RoboDK station: kr30 cnc 101019.rdk

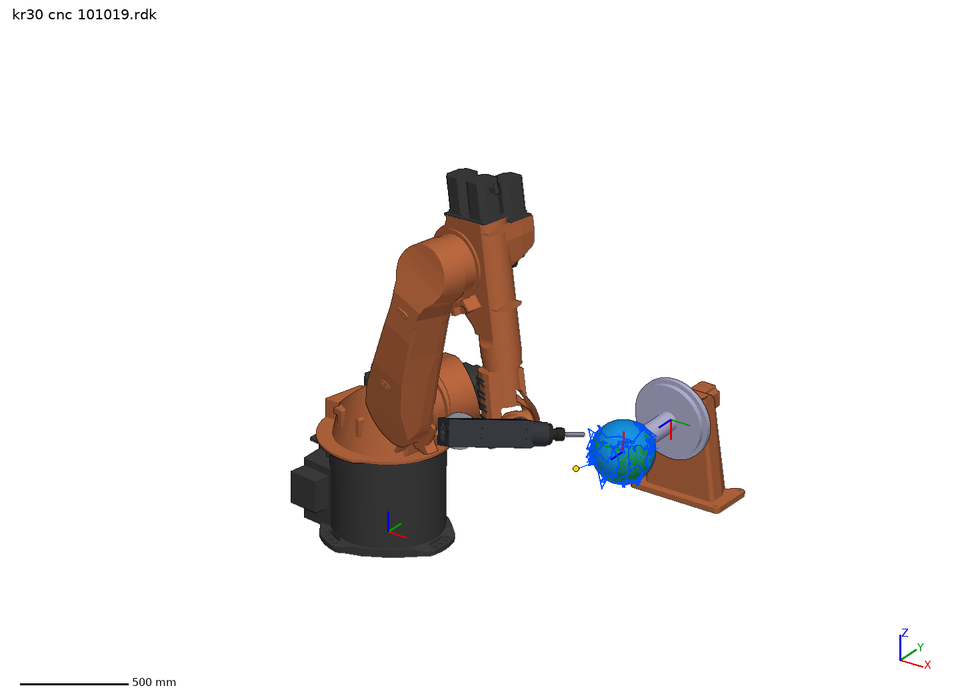
[picture v0: the station drawn from its stored meshes, robots at their saved joint values, targets as dots, program paths as lines]
Station kr30 cnc 101019. Poses are relative to the parent item; angles as X-Y-Z fixed-axis rotations.
  - frame KUKA KR 30 HA Base at (0, 0, 0) mm
    - robot KUKA KR 30 HA: 6 axes, payload 30 kg, reach 2033 mm, repeatability 0.05 mm, weight 665 kg
        modified DH rows (alpha deg, a mm, theta deg, d mm): 0, 0, 0, 815; -90, 350, 0, 0; 0, 850, -90, 0; -90, 145, 0, 820; 90, 0, 0, 0; -90, 0, 180, 170
        joint limits [-185, -135, -120, -350, -119, -350] to [185, 35, 158, 350, 119, 350]; home [0, -90, 90, 0, 0, 0]; saved at [14.33, -73.83, 154.58, -18.35, -102.46, -76.72]
      - tool Spindle, TCP at (249.17, -0.03, 160.93) mm, rotated rx 0 ry 90 rz 0 deg, size 170 x 692.9 x 256 mm
  - frame KUKA KP1 MD250 Base at (1360.87, 339.35, 824.43) mm, rotated rx -93.1 ry 88.62 rz 178.42 deg
    - robot KUKA KP1 MD250: 1 axes, payload 250 kg
        modified DH rows (alpha deg, a mm, theta deg, d mm): 0, 0, 0, 0
        joint limits [-180] to [180]; home [0]; saved at [-180]
      - frame MillingEarth at (0, 0, 402.47) mm
        - object Earth at (0, 0, 0) mm, size 359.7 x 359.7 x 550 mm
  - machining project MillingEarth Settings: C:/Users/albert/Desktop/RoboDK/Deploy/RoboDK_vc2013x64/Library/Milling Earth (5axis).nc | rotZ(0) | rotX(0)*rotY(0) | rotZ(-90)
  - program MillingEarth (2760 instructions, listed below)
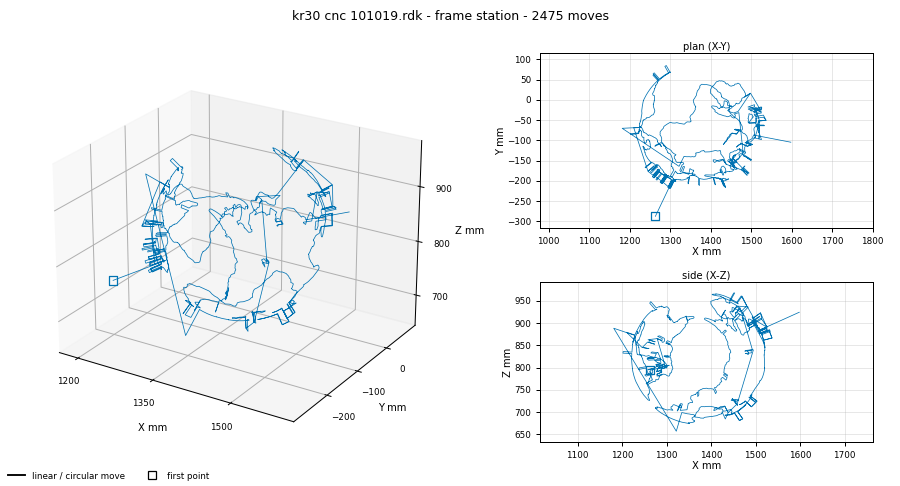
[picture p0: tool path of kr30 cnc 101019.rdk in frame station, 2475 of 2475 moves have a stored position in this frame; points joined in program order, loops and branches not executed]

--- program MillingEarth (robot KUKA KR 30 HA) ---
  Call onMillingEarth_Start
  Set Ref.: MillingEarth
  Set Tool: Spindle
  Show Spindle
  Set speed (1000.0 mm/s)
  MoveJ 1 to (-32.4, 113.46, 221.55) mm, rotated rx 152.37 ry 0 rz 15.09 deg; joints [139.176, -8.287, 13.837, -94.776, 49.407, 99.946, 25, -15.085]
  Set speed (16.7 mm/s)
  Call SetCLW
  Call SetRPM(70.0)
  MoveL 2 to (-32.4, 113.46, 221.55) mm, rotated rx 152.37 ry 0 rz 15.09 deg; joints [139.176, -8.287, 13.837, -94.776, 49.407, 99.946, 25, -15.085]
  Call onMillingEarth_Approach
  MoveL 3 to (-20.33, 68.69, 132.95) mm, rotated rx 152.37 ry 0 rz 15.09 deg; joints [139.274, -8.116, 17.253, -97.785, 49.897, 104.611, 25, -15.085]
  Call onMillingEarth_PathStart
  MoveL 4 to (-20.33, 68.69, 132.95) mm, rotated rx 152.37 ry 0 rz 15.09 deg; joints [139.274, -8.116, 17.253, -97.785, 49.897, 104.611, 25, -15.085]
  MoveL 5 to (-19.96, 69.22, 132.73) mm, rotated rx 152.2 ry 0 rz 14.7 deg; joints [139.228, -8.19, 17.323, -97.794, 49.851, 104.788, 25, -14.701]
  Set speed (16.7 mm/s)
  MoveL 6 to (-22.33, 78.24, 150.42) mm, rotated rx 152.2 ry 0 rz 14.7 deg; joints [139.207, -8.249, 16.662, -97.195, 49.737, 103.856, 25, -14.701]
  Set speed (1000.0 mm/s)
  MoveL 7 to (39.62, 97.38, 134.89) mm, rotated rx 142.85 ry 0 rz -22.62 deg; joints [136.549, -12.268, 20.676, -97.886, 47.129, 113.655, 25, 22.621]
  Set speed (5.0 mm/s)
  MoveL 8 to (34.97, 86.23, 118.95) mm, rotated rx 142.85 ry 0 rz -22.62 deg; joints [136.649, -12.102, 21.236, -98.523, 47.331, 114.615, 25, 22.621]
  Set speed (16.7 mm/s)
  MoveL 9 to (35.17, 86.21, 118.9) mm, rotated rx 142.83 ry 0 rz -22.74 deg; joints [136.641, -12.113, 21.248, -98.526, 47.324, 114.645, 25, 22.74]
  MoveL 10 to (35.37, 86.18, 118.87) mm, rotated rx 142.83 ry 0 rz -22.74 deg; joints [136.645, -12.121, 21.255, -98.524, 47.327, 114.643, 25, 22.74]
  MoveL 11 to (39.2, 85.43, 118.2) mm, rotated rx 142.42 ry 0 rz -25.07 deg; joints [136.528, -12.284, 21.429, -98.569, 47.214, 115.088, 25, 25.069]
  Set speed (16.7 mm/s)
  MoveL 12 to (44.37, 96.48, 134.05) mm, rotated rx 142.42 ry 0 rz -25.07 deg; joints [136.424, -12.455, 20.874, -97.931, 47.008, 114.127, 25, 25.069]
  Set speed (1000.0 mm/s)
  MoveL 13 to (45.45, 92.09, 136.75) mm, rotated rx 142.45 ry 0 rz -25.38 deg; joints [136.592, -12.373, 20.769, -97.864, 47.17, 114.031, 25, 25.381]
  Set speed (5.0 mm/s)
  MoveL 14 to (40.23, 81.08, 120.9) mm, rotated rx 142.45 ry 0 rz -25.38 deg; joints [136.696, -12.202, 21.325, -98.499, 47.375, 114.99, 25, 25.381]
  Set speed (16.7 mm/s)
  MoveL 15 to (37.93, 80.72, 121.87) mm, rotated rx 143.08 ry 0 rz -24.14 deg; joints [136.875, -11.951, 21.058, -98.432, 47.548, 114.307, 25, 24.137]
  MoveL 16 to (37.59, 80.7, 121.99) mm, rotated rx 143.15 ry 0 rz -23.96 deg; joints [136.894, -11.922, 21.028, -98.425, 47.566, 114.235, 25, 23.959]
  MoveL 17 to (35.64, 80.36, 122.79) mm, rotated rx 143.67 ry 0 rz -22.88 deg; joints [137.044, -11.71, 20.804, -98.371, 47.711, 113.664, 25, 22.88]
  MoveL 18 to (35.2, 80.32, 122.95) mm, rotated rx 143.67 ry 0 rz -22.88 deg; joints [137.041, -11.689, 20.785, -98.374, 47.708, 113.667, 25, 22.88]
  MoveL 19 to (34.17, 80.49, 123.13) mm, rotated rx 143.67 ry 0 rz -22.88 deg; joints [137.022, -11.648, 20.748, -98.383, 47.69, 113.677, 25, 22.88]
  MoveL 20 to (33.97, 80.56, 123.14) mm, rotated rx 143.68 ry 0 rz -22.74 deg; joints [137.024, -11.645, 20.745, -98.383, 47.692, 113.67, 25, 22.74]
  MoveL 21 to (33.46, 80.79, 123.13) mm, rotated rx 143.68 ry 0 rz -22.74 deg; joints [137.009, -11.628, 20.731, -98.389, 47.678, 113.677, 25, 22.74]
  MoveL 22 to (32.55, 81.6, 122.84) mm, rotated rx 143.68 ry 0 rz -22.74 deg; joints [136.969, -11.608, 20.718, -98.407, 47.64, 113.694, 25, 22.74]
  MoveL 23 to (31.58, 82.93, 122.2) mm, rotated rx 143.26 ry 0 rz -21.82 deg; joints [136.85, -11.777, 20.895, -98.45, 47.525, 114.146, 25, 21.82]
  MoveL 24 to (31.06, 83.97, 121.62) mm, rotated rx 143.25 ry 0 rz -21.8 deg; joints [136.804, -11.787, 20.912, -98.469, 47.481, 114.18, 25, 21.796]
  MoveL 25 to (31.07, 84.77, 121.06) mm, rotated rx 143.23 ry 0 rz -21.78 deg; joints [136.773, -11.813, 20.942, -98.481, 47.452, 114.203, 25, 21.777]
  MoveL 26 to (31.31, 85.29, 120.63) mm, rotated rx 143.22 ry 0 rz -21.76 deg; joints [136.756, -11.841, 20.971, -98.488, 47.435, 114.217, 25, 21.764]
  MoveL 27 to (31.95, 85.85, 120.07) mm, rotated rx 143.21 ry 0 rz -21.74 deg; joints [136.742, -11.889, 21.018, -98.492, 47.421, 114.232, 25, 21.744]
  MoveL 28 to (32.84, 86.09, 119.65) mm, rotated rx 143.2 ry 0 rz -21.73 deg; joints [136.742, -11.94, 21.067, -98.489, 47.421, 114.241, 25, 21.725]
  MoveL 29 to (34.47, 86.24, 119.09) mm, rotated rx 142.85 ry 0 rz -22.62 deg; joints [136.643, -12.079, 21.216, -98.527, 47.325, 114.619, 25, 22.621]
  Set speed (16.7 mm/s)
  MoveL 30 to (39.12, 97.38, 135.03) mm, rotated rx 142.85 ry 0 rz -22.62 deg; joints [136.543, -12.246, 20.655, -97.89, 47.124, 113.659, 25, 22.621]
  Set speed (1000.0 mm/s)
  MoveL 31 to (36.17, 117.37, 119.01) mm, rotated rx 134.2 ry 0 rz -15.97 deg; joints [134.05, -15.758, 24.592, -99.02, 44.748, 123.399, 25, 15.969]
  Set speed (5.0 mm/s)
  MoveL 32 to (32.22, 103.58, 105.07) mm, rotated rx 134.2 ry 0 rz -15.97 deg; joints [134.235, -15.494, 25.053, -99.679, 45.046, 124.37, 25, 15.969]
  Set speed (16.7 mm/s)
  MoveL 33 to (31.89, 100.84, 107.81) mm, rotated rx 135.66 ry 0 rz -16.2 deg; joints [134.674, -14.947, 24.398, -99.43, 45.455, 122.657, 25, 16.204]
  Set speed (16.7 mm/s)
  MoveL 34 to (35.79, 114.26, 122.11) mm, rotated rx 135.66 ry 0 rz -16.2 deg; joints [134.504, -15.195, 23.92, -98.774, 45.174, 121.686, 25, 16.204]
  Set speed (1000.0 mm/s)
  MoveL 35 to (30.39, 115.24, 122.65) mm, rotated rx 135.75 ry 0 rz -15.97 deg; joints [134.416, -14.981, 23.732, -98.826, 45.093, 121.659, 25, 15.969]
  Set speed (5.0 mm/s)
  MoveL 36 to (26.55, 101.82, 108.33) mm, rotated rx 135.75 ry 0 rz -15.97 deg; joints [134.585, -14.735, 24.211, -99.483, 45.373, 122.63, 25, 15.969]
  Set speed (16.7 mm/s)
  MoveL 37 to (26.92, 104.59, 105.56) mm, rotated rx 134.26 ry 0 rz -15.75 deg; joints [134.14, -15.29, 24.877, -99.738, 44.958, 124.377, 25, 15.751]
  Set speed (16.7 mm/s)
  MoveL 38 to (30.8, 118.38, 119.52) mm, rotated rx 134.26 ry 0 rz -15.75 deg; joints [133.955, -15.553, 24.415, -99.078, 44.66, 123.405, 25, 15.751]
  Set speed (1000.0 mm/s)
  MoveL 39 to (18.54, 129.47, 110.19) mm, rotated rx 130.91 ry 0 rz -8.51 deg; joints [132.886, -16.936, 26.108, -99.738, 43.669, 127.441, 25, 8.507]
  Set speed (5.0 mm/s)
  MoveL 40 to (16.3, 114.52, 97.09) mm, rotated rx 130.91 ry 0 rz -8.51 deg; joints [133.106, -16.636, 26.53, -100.402, 44.009, 128.412, 25, 8.507]
  Set speed (16.7 mm/s)
  MoveL 41 to (17.17, 114.58, 96.87) mm, rotated rx 130.8 ry 0 rz -8.93 deg; joints [133.073, -16.676, 26.58, -100.425, 43.979, 128.547, 25, 8.927]
  MoveL 42 to (17.11, 114.6, 96.86) mm, rotated rx 128.95 ry 0 rz -8.37 deg; joints [132.658, -17.221, 27.272, -100.725, 43.604, 130.708, 25, 8.369]
  MoveL 43 to (16.23, 114.67, 96.93) mm, rotated rx 128.98 ry 0 rz -7.94 deg; joints [132.668, -17.209, 27.257, -100.717, 43.613, 130.666, 25, 7.936]
  Set speed (16.7 mm/s)
  MoveL 44 to (18.38, 130.06, 109.51) mm, rotated rx 128.98 ry 0 rz -7.94 deg; joints [132.428, -17.529, 26.858, -100.056, 43.251, 129.7, 25, 7.936]
  Set speed (1000.0 mm/s)
  MoveL 45 to (51.72, 163.01, 1.41) mm, rotated rx 91.23 ry 0 rz -17.25 deg; joints [121.681, -25.825, 44.795, -117.777, 36.413, 186.971, 25, 17.255]
  Set speed (5.0 mm/s)
  MoveL 46 to (45.79, 143.91, 0.98) mm, rotated rx 91.23 ry 0 rz -17.25 deg; joints [122.333, -25.195, 44.709, -117.822, 37.21, 187.295, 25, 17.255]
  Set speed (16.7 mm/s)
  MoveL 47 to (46.25, 143.76, 1.2) mm, rotated rx 91.32 ry 0 rz -17.44 deg; joints [122.349, -25.193, 44.674, -117.768, 37.209, 187.15, 25, 17.439]
  MoveL 48 to (46.82, 143.57, 1.59) mm, rotated rx 91.32 ry 0 rz -17.44 deg; joints [122.369, -25.22, 44.679, -117.724, 37.215, 187.104, 25, 17.439]
  MoveL 49 to (49.93, 142.45, 4.46) mm, rotated rx 92.41 ry 0 rz -18.69 deg; joints [122.588, -25.183, 44.214, -117.028, 37.202, 185.23, 25, 18.692]
  MoveL 50 to (49.93, 142.46, 4.45) mm, rotated rx 92.58 ry 0 rz -18.98 deg; joints [122.597, -25.142, 44.135, -116.974, 37.192, 184.997, 25, 18.983]
  MoveL 51 to (53.02, 141.29, 5.69) mm, rotated rx 93.05 ry 0 rz -20.24 deg; joints [122.693, -25.121, 43.934, -116.677, 37.192, 184.195, 25, 20.235]
  MoveL 52 to (53.52, 141.09, 5.97) mm, rotated rx 93.05 ry 0 rz -20.24 deg; joints [122.71, -25.145, 43.94, -116.641, 37.198, 184.157, 25, 20.235]
  MoveL 53 to (54.32, 140.74, 7.02) mm, rotated rx 93.05 ry 0 rz -20.24 deg; joints [122.748, -25.181, 43.93, -116.553, 37.21, 184.062, 25, 20.235]
  MoveL 54 to (54.41, 140.69, 7.24) mm, rotated rx 93.13 ry 0 rz -20.27 deg; joints [122.765, -25.177, 43.894, -116.501, 37.21, 183.92, 25, 20.271]
  MoveL 55 to (54.58, 140.57, 8.16) mm, rotated rx 93.13 ry 0 rz -20.27 deg; joints [122.786, -25.183, 43.868, -116.446, 37.213, 183.859, 25, 20.271]
  MoveL 56 to (54.59, 140.48, 9.51) mm, rotated rx 93.64 ry 0 rz -20.29 deg; joints [122.893, -25.155, 43.647, -116.124, 37.219, 182.987, 25, 20.287]
  MoveL 57 to (54.58, 140.49, 9.48) mm, rotated rx 94.31 ry 0 rz -20.6 deg; joints [122.985, -25.085, 43.395, -115.828, 37.218, 181.983, 25, 20.6]
  MoveL 58 to (58.8, 138.43, 13.63) mm, rotated rx 95.89 ry 0 rz -22.38 deg; joints [123.331, -24.972, 42.705, -114.851, 37.268, 179.312, 25, 22.379]
  MoveL 59 to (58.75, 138.46, 13.59) mm, rotated rx 96.1 ry 0 rz -22.84 deg; joints [123.338, -24.902, 42.595, -114.798, 37.258, 179.034, 25, 22.841]
  MoveL 60 to (63.19, 136.41, 14.38) mm, rotated rx 96.4 ry 0 rz -24.7 deg; joints [123.405, -24.877, 42.464, -114.615, 37.271, 178.531, 25, 24.703]
  MoveL 61 to (63.44, 136.29, 14.44) mm, rotated rx 96.4 ry 0 rz -24.7 deg; joints [123.413, -24.889, 42.47, -114.601, 37.275, 178.517, 25, 24.703]
  MoveL 62 to (63.67, 136.17, 14.51) mm, rotated rx 96.43 ry 0 rz -24.8 deg; joints [123.419, -24.886, 42.458, -114.585, 37.276, 178.471, 25, 24.802]
  MoveL 63 to (65.41, 135.28, 15.07) mm, rotated rx 96.66 ry 0 rz -25.65 deg; joints [123.465, -24.854, 42.346, -114.453, 37.284, 178.084, 25, 25.652]
  MoveL 64 to (65.72, 135.13, 15.13) mm, rotated rx 96.69 ry 0 rz -25.78 deg; joints [123.47, -24.852, 42.337, -114.44, 37.285, 178.049, 25, 25.782]
  MoveL 65 to (68.28, 133.79, 15.64) mm, rotated rx 96.88 ry 0 rz -26.87 deg; joints [123.515, -24.836, 42.253, -114.321, 37.296, 177.723, 25, 26.869]
  MoveL 66 to (68.86, 133.47, 15.86) mm, rotated rx 96.88 ry 0 rz -26.87 deg; joints [123.535, -24.865, 42.265, -114.285, 37.306, 177.685, 25, 26.869]
  MoveL 67 to (69.74, 132.95, 16.36) mm, rotated rx 97.07 ry 0 rz -27.25 deg; joints [123.578, -24.847, 42.181, -114.171, 37.317, 177.369, 25, 27.255]
  MoveL 68 to (69.89, 132.86, 16.45) mm, rotated rx 97.07 ry 0 rz -27.25 deg; joints [123.584, -24.855, 42.183, -114.159, 37.32, 177.357, 25, 27.255]
  MoveL 69 to (76.53, 128.45, 21.19) mm, rotated rx 98.88 ry 0 rz -30.29 deg; joints [124.008, -24.668, 41.377, -113.079, 37.443, 174.342, 25, 30.29]
  MoveL 70 to (76.49, 128.48, 21.19) mm, rotated rx 98.98 ry 0 rz -31.03 deg; joints [123.98, -24.572, 41.284, -113.105, 37.42, 174.266, 25, 31.033]
  MoveL 71 to (80.12, 126.44, 20.02) mm, rotated rx 98.53 ry 0 rz -32.62 deg; joints [123.873, -24.622, 41.485, -113.371, 37.385, 175.011, 25, 32.625]
  MoveL 72 to (80.83, 126, 19.93) mm, rotated rx 98.53 ry 0 rz -32.62 deg; joints [123.891, -24.66, 41.513, -113.345, 37.397, 174.985, 25, 32.625]
  MoveL 73 to (81.28, 125.71, 19.96) mm, rotated rx 98.54 ry 0 rz -32.83 deg; joints [123.894, -24.658, 41.507, -113.337, 37.398, 174.965, 25, 32.828]
  MoveL 74 to (81.75, 125.39, 20.06) mm, rotated rx 98.54 ry 0 rz -32.83 deg; joints [123.909, -24.682, 41.52, -113.312, 37.407, 174.939, 25, 32.828]
  MoveL 75 to (86.58, 121.8, 21.83) mm, rotated rx 99.22 ry 0 rz -35.13 deg; joints [124.071, -24.606, 41.216, -112.912, 37.46, 173.813, 25, 35.132]
  MoveL 76 to (87.18, 121.32, 22.1) mm, rotated rx 99.31 ry 0 rz -35.38 deg; joints [124.096, -24.601, 41.179, -112.855, 37.469, 173.663, 25, 35.383]
  MoveL 77 to (91.51, 117.76, 23.78) mm, rotated rx 99.97 ry 0 rz -37.57 deg; joints [124.252, -24.518, 40.882, -112.478, 37.525, 172.586, 25, 37.568]
  MoveL 78 to (91.73, 117.56, 23.89) mm, rotated rx 99.97 ry 0 rz -37.57 deg; joints [124.261, -24.53, 40.886, -112.462, 37.53, 172.569, 25, 37.568]
  MoveL 79 to (92.05, 117.28, 24.08) mm, rotated rx 100.04 ry 0 rz -37.73 deg; joints [124.279, -24.521, 40.854, -112.421, 37.537, 172.451, 25, 37.73]
  MoveL 80 to (92.22, 117.12, 24.19) mm, rotated rx 100.04 ry 0 rz -37.73 deg; joints [124.286, -24.53, 40.856, -112.407, 37.541, 172.436, 25, 37.73]
  MoveL 81 to (94.43, 114.96, 25.97) mm, rotated rx 100.72 ry 0 rz -38.91 deg; joints [124.454, -24.442, 40.549, -112.016, 37.607, 171.32, 25, 38.912]
  MoveL 82 to (96.38, 113.21, 26.49) mm, rotated rx 101.03 ry 0 rz -40.21 deg; joints [124.508, -24.372, 40.397, -111.879, 37.625, 170.856, 25, 40.208]
  MoveL 83 to (96.7, 112.9, 26.63) mm, rotated rx 101.03 ry 0 rz -40.21 deg; joints [124.521, -24.39, 40.405, -111.857, 37.633, 170.832, 25, 40.208]
  MoveL 84 to (96.94, 112.66, 26.77) mm, rotated rx 101.08 ry 0 rz -40.34 deg; joints [124.534, -24.382, 40.381, -111.827, 37.638, 170.745, 25, 40.339]
  MoveL 85 to (97.15, 112.45, 26.91) mm, rotated rx 101.08 ry 0 rz -40.34 deg; joints [124.544, -24.394, 40.384, -111.809, 37.644, 170.727, 25, 40.339]
  MoveL 86 to (99.43, 109.95, 28.85) mm, rotated rx 101.83 ry 0 rz -41.63 deg; joints [124.732, -24.29, 40.046, -111.39, 37.725, 169.515, 25, 41.631]
  MoveL 87 to (99.68, 109.66, 29.07) mm, rotated rx 101.92 ry 0 rz -41.79 deg; joints [124.753, -24.277, 40.006, -111.342, 37.735, 169.374, 25, 41.785]
  MoveL 88 to (100.05, 109.21, 29.52) mm, rotated rx 101.92 ry 0 rz -41.79 deg; joints [124.776, -24.296, 40.006, -111.302, 37.748, 169.331, 25, 41.785]
  MoveL 89 to (101.45, 107.18, 32.04) mm, rotated rx 102.89 ry 0 rz -42.72 deg; joints [125.025, -24.151, 39.561, -110.764, 37.865, 167.759, 25, 42.715]
  MoveL 90 to (101.64, 106.86, 32.53) mm, rotated rx 102.89 ry 0 rz -42.72 deg; joints [125.044, -24.16, 39.553, -110.73, 37.876, 167.722, 25, 42.715]
  MoveL 91 to (101.66, 106.43, 33.85) mm, rotated rx 102.89 ry 0 rz -42.72 deg; joints [125.079, -24.156, 39.512, -110.66, 37.895, 167.646, 25, 42.715]
  MoveL 92 to (101.59, 106.39, 34.17) mm, rotated rx 103.02 ry 0 rz -42.71 deg; joints [125.111, -24.137, 39.456, -110.593, 37.91, 167.448, 25, 42.707]
  MoveL 93 to (101.26, 106.41, 35.09) mm, rotated rx 103.02 ry 0 rz -42.71 deg; joints [125.125, -24.114, 39.413, -110.56, 37.916, 167.411, 25, 42.707]
  MoveL 94 to (100.18, 106.74, 37.1) mm, rotated rx 103.8 ry 0 rz -42.31 deg; joints [125.33, -23.987, 39.054, -110.139, 38.02, 166.158, 25, 42.306]
  MoveL 95 to (100.18, 106.75, 37.07) mm, rotated rx 104.74 ry 0 rz -42.37 deg; joints [125.518, -23.857, 38.713, -109.758, 38.119, 164.802, 25, 42.369]
  MoveL 96 to (101.87, 103.05, 42.54) mm, rotated rx 107.02 ry 0 rz -43.96 deg; joints [126.117, -23.434, 37.664, -108.618, 38.461, 161.255, 25, 43.965]
  MoveL 97 to (102.05, 102.73, 42.88) mm, rotated rx 107.16 ry 0 rz -44.1 deg; joints [126.154, -23.408, 37.602, -108.551, 38.484, 161.046, 25, 44.103]
  MoveL 98 to (104.05, 99.2, 46.26) mm, rotated rx 108.54 ry 0 rz -45.69 deg; joints [126.529, -23.131, 36.964, -107.889, 38.717, 158.936, 25, 45.694]
  MoveL 99 to (104.28, 98.54, 47.15) mm, rotated rx 108.59 ry 0 rz -45.69 deg; joints [126.576, -23.134, 36.93, -107.816, 38.749, 158.809, 25, 45.689]
  MoveL 100 to (104.13, 98.18, 48.22) mm, rotated rx 108.63 ry 0 rz -45.69 deg; joints [126.616, -23.114, 36.875, -107.75, 38.775, 158.69, 25, 45.685]
  MoveL 101 to (103.98, 98.01, 48.88) mm, rotated rx 108.9 ry 0 rz -45.69 deg; joints [126.69, -23.059, 36.751, -107.625, 38.823, 158.286, 25, 45.689]
  MoveL 102 to (103.97, 98.04, 48.86) mm, rotated rx 109.5 ry 0 rz -45.93 deg; joints [126.807, -22.933, 36.514, -107.423, 38.898, 157.459, 25, 45.928]
  MoveL 103 to (104.32, 97.19, 49.77) mm, rotated rx 109.87 ry 0 rz -46.27 deg; joints [126.911, -22.854, 36.343, -107.253, 38.966, 156.903, 25, 46.27]
  MoveL 104 to (104.27, 97.22, 49.84) mm, rotated rx 109.04 ry 0 rz -47.98 deg; joints [126.625, -22.816, 36.523, -107.68, 38.767, 158.195, 25, 47.98]
  MoveL 105 to (104.53, 98.86, 45.91) mm, rotated rx 107.47 ry 0 rz -47.56 deg; joints [126.189, -23.136, 37.252, -108.436, 38.492, 160.603, 25, 47.562]
  MoveL 106 to (104.48, 99.07, 45.58) mm, rotated rx 107.19 ry 0 rz -47.43 deg; joints [126.126, -23.189, 37.369, -108.552, 38.453, 161.005, 25, 47.435]
  MoveL 107 to (104.22, 100.62, 42.67) mm, rotated rx 106.04 ry 0 rz -46.91 deg; joints [125.812, -23.408, 37.902, -109.131, 38.267, 162.8, 25, 46.913]
  Set speed (16.7 mm/s)
  MoveL 108 to (118.26, 113.75, 48.19) mm, rotated rx 106.04 ry 0 rz -46.91 deg; joints [125.309, -23.945, 37.793, -108.673, 37.596, 162.064, 25, 46.913]
  Set speed (1000.0 mm/s)
  MoveL 109 to (121.75, 111.27, 45.2) mm, rotated rx 106.02 ry 0 rz -47.09 deg; joints [125.325, -24.149, 38.019, -108.689, 37.618, 162.103, 25, 47.094]
  Set speed (5.0 mm/s)
  MoveL 110 to (107.67, 98.18, 39.68) mm, rotated rx 106.02 ry 0 rz -47.09 deg; joints [125.829, -23.611, 38.128, -109.147, 38.29, 162.841, 25, 47.094]
  Set speed (16.7 mm/s)
  MoveL 111 to (109.17, 95.75, 41.47) mm, rotated rx 106.73 ry 0 rz -48.2 deg; joints [126.02, -23.479, 37.802, -108.791, 38.402, 161.741, 25, 48.199]
  MoveL 112 to (109.28, 95.57, 41.61) mm, rotated rx 106.78 ry 0 rz -48.28 deg; joints [126.034, -23.469, 37.778, -108.764, 38.411, 161.658, 25, 48.282]
  MoveL 113 to (110.67, 92.99, 43.73) mm, rotated rx 107.58 ry 0 rz -49.35 deg; joints [126.258, -23.32, 37.409, -108.361, 38.547, 160.415, 25, 49.349]
  MoveL 114 to (110.84, 92.61, 44.1) mm, rotated rx 107.58 ry 0 rz -49.35 deg; joints [126.277, -23.33, 37.405, -108.333, 38.559, 160.385, 25, 49.349]
  MoveL 115 to (110.92, 91.99, 45.19) mm, rotated rx 107.58 ry 0 rz -49.35 deg; joints [126.315, -23.333, 37.377, -108.272, 38.584, 160.319, 25, 49.349]
  MoveL 116 to (110.89, 91.91, 45.44) mm, rotated rx 107.68 ry 0 rz -49.37 deg; joints [126.341, -23.314, 37.332, -108.225, 38.601, 160.17, 25, 49.367]
  MoveL 117 to (110.71, 91.74, 46.19) mm, rotated rx 107.68 ry 0 rz -49.37 deg; joints [126.359, -23.302, 37.303, -108.194, 38.612, 160.136, 25, 49.367]
  MoveL 118 to (110.22, 91.6, 47.62) mm, rotated rx 108.25 ry 0 rz -49.28 deg; joints [126.518, -23.185, 37.037, -107.918, 38.712, 159.256, 25, 49.281]
  MoveL 119 to (110.22, 91.62, 47.57) mm, rotated rx 109.14 ry 0 rz -49.7 deg; joints [126.686, -22.998, 36.684, -107.62, 38.817, 158.035, 25, 49.698]
  MoveL 120 to (112.14, 87.75, 50.32) mm, rotated rx 110.24 ry 0 rz -51.38 deg; joints [126.995, -22.762, 36.173, -107.111, 39.022, 156.374, 25, 51.383]
  MoveL 121 to (112.4, 86.84, 51.32) mm, rotated rx 110.24 ry 0 rz -51.38 deg; joints [127.041, -22.778, 36.157, -107.046, 39.055, 156.305, 25, 51.383]
  MoveL 122 to (112.13, 86.41, 52.6) mm, rotated rx 110.24 ry 0 rz -51.38 deg; joints [127.076, -22.761, 36.111, -106.991, 39.079, 156.245, 25, 51.383]
  MoveL 123 to (112.01, 86.37, 52.93) mm, rotated rx 110.38 ry 0 rz -51.36 deg; joints [127.114, -22.731, 36.048, -106.931, 39.105, 156.045, 25, 51.361]
  MoveL 124 to (111.32, 86.54, 54.09) mm, rotated rx 110.38 ry 0 rz -51.36 deg; joints [127.128, -22.686, 35.986, -106.903, 39.113, 156.012, 25, 51.361]
  MoveL 125 to (110.56, 86.95, 54.96) mm, rotated rx 110.73 ry 0 rz -51.04 deg; joints [127.23, -22.606, 35.82, -106.743, 39.183, 155.479, 25, 51.039]
  MoveL 126 to (110.59, 86.95, 54.91) mm, rotated rx 111.91 ry 0 rz -51.03 deg; joints [127.496, -22.394, 35.39, -106.336, 39.369, 153.85, 25, 51.03]
  MoveL 127 to (110.98, 85.3, 56.68) mm, rotated rx 112.64 ry 0 rz -51.65 deg; joints [127.704, -22.223, 35.052, -106.026, 39.517, 152.785, 25, 51.653]
  MoveL 128 to (111.01, 84.82, 57.35) mm, rotated rx 112.64 ry 0 rz -51.65 deg; joints [127.731, -22.225, 35.036, -105.99, 39.537, 152.746, 25, 51.653]
  MoveL 129 to (110.99, 84.64, 57.66) mm, rotated rx 112.76 ry 0 rz -51.7 deg; joints [127.767, -22.195, 34.977, -105.937, 39.564, 152.561, 25, 51.701]
  MoveL 130 to (110.91, 84.43, 58.11) mm, rotated rx 112.76 ry 0 rz -51.7 deg; joints [127.782, -22.19, 34.961, -105.917, 39.574, 152.539, 25, 51.701]
  MoveL 131 to (110.03, 83.05, 61.67) mm, rotated rx 114.23 ry 0 rz -51.92 deg; joints [128.21, -21.827, 34.274, -105.313, 39.89, 150.405, 25, 51.923]
  MoveL 132 to (109.88, 82.88, 62.17) mm, rotated rx 114.4 ry 0 rz -51.94 deg; joints [128.26, -21.784, 34.195, -105.244, 39.927, 150.169, 25, 51.938]
  MoveL 133 to (109.06, 81.95, 64.77) mm, rotated rx 115.48 ry 0 rz -52.03 deg; joints [128.579, -21.504, 33.689, -104.82, 40.169, 148.622, 25, 52.033]
  MoveL 134 to (109.07, 81.98, 64.73) mm, rotated rx 116.1 ry 0 rz -52.39 deg; joints [128.701, -21.342, 33.437, -104.655, 40.262, 147.815, 25, 52.385]
  MoveL 135 to (109.68, 79.86, 66.33) mm, rotated rx 116.77 ry 0 rz -53.25 deg; joints [128.9, -21.163, 33.124, -104.404, 40.417, 146.871, 25, 53.249]
  MoveL 136 to (109.69, 79.87, 66.3) mm, rotated rx 116.91 ry 0 rz -53.52 deg; joints [128.916, -21.109, 33.055, -104.38, 40.429, 146.701, 25, 53.52]
  MoveL 137 to (110.88, 77.27, 67.41) mm, rotated rx 117.38 ry 0 rz -54.7 deg; joints [129.055, -20.983, 32.838, -104.209, 40.538, 146.049, 25, 54.699]
  MoveL 138 to (111.03, 76.87, 67.61) mm, rotated rx 117.38 ry 0 rz -54.7 deg; joints [129.071, -20.994, 32.841, -104.192, 40.551, 146.032, 25, 54.699]
  MoveL 139 to (111.15, 76.07, 68.3) mm, rotated rx 117.38 ry 0 rz -54.7 deg; joints [129.108, -21.004, 32.831, -104.151, 40.581, 145.988, 25, 54.699]
  MoveL 140 to (111.14, 75.85, 68.56) mm, rotated rx 117.49 ry 0 rz -54.77 deg; joints [129.141, -20.974, 32.78, -104.111, 40.607, 145.835, 25, 54.773]
  MoveL 141 to (111.07, 75.48, 69.1) mm, rotated rx 117.49 ry 0 rz -54.77 deg; joints [129.161, -20.97, 32.764, -104.088, 40.624, 145.809, 25, 54.773]
  MoveL 142 to (110.3, 73.8, 72.07) mm, rotated rx 118.76 ry 0 rz -55.17 deg; joints [129.543, -20.613, 32.169, -103.639, 40.929, 144.045, 25, 55.173]
  MoveL 143 to (110.19, 73.63, 72.41) mm, rotated rx 118.76 ry 0 rz -55.17 deg; joints [129.554, -20.607, 32.156, -103.626, 40.939, 144.031, 25, 55.173]
  MoveL 144 to (110.02, 73.45, 72.86) mm, rotated rx 118.95 ry 0 rz -55.2 deg; joints [129.612, -20.551, 32.066, -103.56, 40.986, 143.765, 25, 55.197]
  MoveL 145 to (109.94, 73.37, 73.05) mm, rotated rx 118.95 ry 0 rz -55.2 deg; joints [129.618, -20.547, 32.058, -103.554, 40.99, 143.758, 25, 55.197]
  MoveL 146 to (108.02, 71.92, 77.24) mm, rotated rx 120.78 ry 0 rz -55.24 deg; joints [130.169, -20.011, 31.204, -102.95, 41.444, 141.27, 25, 55.241]
  MoveL 147 to (107.85, 71.77, 77.62) mm, rotated rx 120.99 ry 0 rz -55.26 deg; joints [130.229, -19.952, 31.112, -102.888, 41.493, 140.998, 25, 55.256]
  MoveL 148 to (105.63, 70.25, 81.94) mm, rotated rx 122.86 ry 0 rz -55.24 deg; joints [130.8, -19.375, 30.235, -102.313, 41.975, 138.502, 25, 55.242]
  MoveL 149 to (104.84, 70.16, 83.03) mm, rotated rx 122.86 ry 0 rz -55.24 deg; joints [130.823, -19.329, 30.176, -102.29, 41.994, 138.477, 25, 55.242]
  MoveL 150 to (104.53, 70.23, 83.36) mm, rotated rx 123.01 ry 0 rz -55.13 deg; joints [130.867, -19.283, 30.108, -102.247, 42.032, 138.283, 25, 55.134]
  MoveL 151 to (104.24, 70.33, 83.64) mm, rotated rx 123.01 ry 0 rz -55.13 deg; joints [130.869, -19.265, 30.089, -102.244, 42.034, 138.28, 25, 55.134]
  MoveL 152 to (101.64, 71.39, 85.9) mm, rotated rx 124.05 ry 0 rz -54.05 deg; joints [131.187, -18.936, 29.605, -101.947, 42.306, 136.916, 25, 54.046]
  MoveL 153 to (101.65, 71.39, 85.9) mm, rotated rx 124.25 ry 0 rz -53.89 deg; joints [131.242, -18.899, 29.543, -101.896, 42.355, 136.664, 25, 53.889]
  MoveL 154 to (99.95, 71.26, 87.98) mm, rotated rx 125.31 ry 0 rz -53.41 deg; joints [131.562, -18.566, 29.064, -101.612, 42.633, 135.296, 25, 53.414]
  MoveL 155 to (99.56, 71.29, 88.39) mm, rotated rx 125.31 ry 0 rz -53.41 deg; joints [131.568, -18.543, 29.038, -101.606, 42.638, 135.289, 25, 53.414]
  MoveL 156 to (99.1, 71.39, 88.83) mm, rotated rx 125.52 ry 0 rz -53.25 deg; joints [131.632, -18.476, 28.942, -101.551, 42.693, 135.023, 25, 53.249]
  MoveL 157 to (98.75, 71.49, 89.13) mm, rotated rx 125.52 ry 0 rz -53.25 deg; joints [131.633, -18.455, 28.921, -101.549, 42.694, 135.021, 25, 53.249]
  MoveL 158 to (93.79, 73.31, 92.93) mm, rotated rx 127.33 ry 0 rz -51.11 deg; joints [132.187, -17.852, 28.085, -101.09, 43.183, 132.714, 25, 51.111]
  MoveL 159 to (93.53, 73.39, 93.13) mm, rotated rx 127.55 ry 0 rz -50.88 deg; joints [132.252, -17.795, 28.002, -101.038, 43.241, 132.438, 25, 50.878]
  MoveL 160 to (88.83, 73.91, 97.23) mm, rotated rx 129.57 ry 0 rz -49.19 deg; joints [132.865, -17.103, 27.081, -100.575, 43.791, 129.933, 25, 49.194]
  MoveL 161 to (88.79, 73.91, 97.27) mm, rotated rx 129.72 ry 0 rz -49.09 deg; joints [132.908, -17.065, 27.028, -100.544, 43.83, 129.745, 25, 49.091]
  MoveL 162 to (87.4, 73.49, 98.82) mm, rotated rx 130.61 ry 0 rz -48.74 deg; joints [133.172, -16.765, 26.638, -100.358, 44.07, 128.665, 25, 48.742]
  MoveL 163 to (87.43, 73.5, 98.79) mm, rotated rx 131.37 ry 0 rz -48.88 deg; joints [133.345, -16.544, 26.361, -100.24, 44.227, 127.783, 25, 48.882]
  MoveL 164 to (87.12, 70.77, 101.04) mm, rotated rx 132.5 ry 0 rz -49.82 deg; joints [133.688, -16.137, 25.848, -100.014, 44.541, 126.418, 25, 49.825]
  MoveL 165 to (86.99, 70.33, 101.45) mm, rotated rx 132.5 ry 0 rz -49.82 deg; joints [133.708, -16.13, 25.835, -100.001, 44.56, 126.404, 25, 49.825]
  MoveL 166 to (86.3, 69.7, 102.47) mm, rotated rx 132.5 ry 0 rz -49.82 deg; joints [133.743, -16.09, 25.785, -99.979, 44.591, 126.382, 25, 49.825]
  MoveL 167 to (86.12, 69.64, 102.67) mm, rotated rx 132.6 ry 0 rz -49.79 deg; joints [133.774, -16.053, 25.739, -99.96, 44.62, 126.259, 25, 49.788]
  MoveL 168 to (85.06, 69.65, 103.54) mm, rotated rx 132.6 ry 0 rz -49.79 deg; joints [133.785, -15.995, 25.677, -99.953, 44.63, 126.252, 25, 49.788]
  MoveL 169 to (83.74, 70.04, 104.35) mm, rotated rx 133.03 ry 0 rz -49.18 deg; joints [133.914, -15.839, 25.485, -99.872, 44.749, 125.741, 25, 49.18]
  MoveL 170 to (83.76, 70.05, 104.32) mm, rotated rx 133.57 ry 0 rz -48.8 deg; joints [134.061, -15.708, 25.313, -99.783, 44.885, 125.108, 25, 48.795]
  MoveL 171 to (82.94, 69.61, 105.27) mm, rotated rx 134.23 ry 0 rz -48.67 deg; joints [134.249, -15.478, 25.033, -99.67, 45.059, 124.334, 25, 48.674]
  MoveL 172 to (82.78, 69.45, 105.51) mm, rotated rx 134.36 ry 0 rz -48.68 deg; joints [134.287, -15.431, 24.976, -99.648, 45.095, 124.185, 25, 48.68]
  MoveL 173 to (81.07, 67.48, 108.08) mm, rotated rx 135.8 ry 0 rz -48.88 deg; joints [134.715, -14.896, 24.337, -99.407, 45.493, 122.5, 25, 48.876]
  Set speed (16.7 mm/s)
  MoveL 174 to (91.57, 76.65, 122.42) mm, rotated rx 135.8 ry 0 rz -48.88 deg; joints [134.546, -15.141, 23.857, -98.752, 45.215, 121.53, 25, 48.876]
  Set speed (1000.0 mm/s)
  MoveL 175 to (90.79, 72.41, 125.54) mm, rotated rx 137.12 ry 0 rz -50.2 deg; joints [134.966, -14.607, 23.235, -98.542, 45.611, 120.003, 25, 50.204]
  Set speed (5.0 mm/s)
  MoveL 176 to (80.33, 63.7, 110.89) mm, rotated rx 137.12 ry 0 rz -50.2 deg; joints [135.121, -14.376, 23.73, -99.194, 45.875, 120.971, 25, 50.204]
  Set speed (16.7 mm/s)
  MoveL 177 to (78.54, 62.71, 112.72) mm, rotated rx 138.15 ry 0 rz -49.98 deg; joints [135.428, -13.977, 23.272, -99.042, 46.165, 119.787, 25, 49.98]
  MoveL 178 to (77.97, 61.99, 113.51) mm, rotated rx 138.89 ry 0 rz -50.1 deg; joints [135.626, -13.715, 22.976, -98.948, 46.352, 118.964, 25, 50.095]
  MoveL 179 to (77.39, 61.55, 114.14) mm, rotated rx 138.89 ry 0 rz -50.1 deg; joints [135.648, -13.684, 22.941, -98.938, 46.373, 118.955, 25, 50.095]
  MoveL 180 to (77.25, 61.49, 114.27) mm, rotated rx 138.96 ry 0 rz -50.07 deg; joints [135.67, -13.654, 22.908, -98.927, 46.394, 118.869, 25, 50.068]
  MoveL 181 to (76.96, 61.41, 114.51) mm, rotated rx 138.96 ry 0 rz -50.07 deg; joints [135.676, -13.639, 22.892, -98.925, 46.4, 118.867, 25, 50.068]
  MoveL 182 to (76.39, 61.28, 114.96) mm, rotated rx 139.22 ry 0 rz -49.91 deg; joints [135.753, -13.537, 22.777, -98.89, 46.473, 118.571, 25, 49.906]
  MoveL 183 to (76.36, 61.31, 114.96) mm, rotated rx 140.09 ry 0 rz -50 deg; joints [135.946, -13.265, 22.476, -98.804, 46.657, 117.63, 25, 50.004]
  MoveL 184 to (75.89, 58.95, 116.5) mm, rotated rx 140.99 ry 0 rz -50.89 deg; joints [136.21, -12.908, 22.084, -98.691, 46.909, 116.625, 25, 50.89]
  MoveL 185 to (75.88, 58.99, 116.48) mm, rotated rx 141.42 ry 0 rz -51.97 deg; joints [136.26, -12.717, 21.891, -98.674, 46.957, 116.184, 25, 51.972]
  MoveL 186 to (78.23, 55.19, 116.8) mm, rotated rx 141.6 ry 0 rz -54.63 deg; joints [136.314, -12.643, 21.81, -98.652, 47.009, 115.978, 25, 54.632]
  MoveL 187 to (78.45, 54.73, 116.87) mm, rotated rx 141.6 ry 0 rz -54.63 deg; joints [136.329, -12.655, 21.819, -98.645, 47.023, 115.97, 25, 54.632]
  MoveL 188 to (78.6, 54.34, 116.95) mm, rotated rx 141.65 ry 0 rz -54.87 deg; joints [136.343, -12.636, 21.798, -98.639, 47.037, 115.916, 25, 54.874]
  MoveL 189 to (78.73, 53.86, 117.08) mm, rotated rx 141.65 ry 0 rz -54.87 deg; joints [136.36, -12.644, 21.803, -98.631, 47.053, 115.908, 25, 54.874]
  MoveL 190 to (79.04, 52.14, 117.64) mm, rotated rx 141.99 ry 0 rz -55.82 deg; joints [136.459, -12.508, 21.656, -98.592, 47.148, 115.532, 25, 55.824]
  MoveL 191 to (79, 52.2, 117.64) mm, rotated rx 141.9 ry 0 rz -57.52 deg; joints [136.365, -12.447, 21.613, -98.636, 47.058, 115.673, 25, 57.524]
  MoveL 192 to (80.03, 51.74, 117.15) mm, rotated rx 141.6 ry 0 rz -58.08 deg; joints [136.28, -12.564, 21.74, -98.671, 46.977, 115.997, 25, 58.085]
  MoveL 193 to (80.55, 51.42, 116.94) mm, rotated rx 141.6 ry 0 rz -58.08 deg; joints [136.286, -12.593, 21.767, -98.667, 46.982, 115.993, 25, 58.085]
  MoveL 194 to (80.84, 51.2, 116.84) mm, rotated rx 141.54 ry 0 rz -58.29 deg; joints [136.268, -12.617, 21.792, -98.674, 46.966, 116.058, 25, 58.287]
  MoveL 195 to (81.31, 50.73, 116.71) mm, rotated rx 141.54 ry 0 rz -58.29 deg; joints [136.28, -12.644, 21.816, -98.668, 46.977, 116.052, 25, 58.287]
  MoveL 196 to (83.31, 48.21, 116.37) mm, rotated rx 141.34 ry 0 rz -60.19 deg; joints [136.222, -12.723, 21.903, -98.692, 46.921, 116.274, 25, 60.191]
  MoveL 197 to (83.12, 48.42, 116.42) mm, rotated rx 141.33 ry 0 rz -60.29 deg; joints [136.209, -12.711, 21.894, -98.698, 46.909, 116.294, 25, 60.286]
  MoveL 198 to (83.31, 48.23, 116.36) mm, rotated rx 141.29 ry 0 rz -60.44 deg; joints [136.2, -12.725, 21.909, -98.702, 46.9, 116.332, 25, 60.436]
  MoveL 199 to (85.09, 46.58, 115.75) mm, rotated rx 140.91 ry 0 rz -61.88 deg; joints [136.086, -12.871, 22.07, -98.75, 46.791, 116.76, 25, 61.878]
  MoveL 200 to (85.39, 46.24, 115.66) mm, rotated rx 140.91 ry 0 rz -61.88 deg; joints [136.094, -12.89, 22.087, -98.746, 46.798, 116.755, 25, 61.878]
  MoveL 201 to (85.89, 45.32, 115.66) mm, rotated rx 140.91 ry 0 rz -61.88 deg; joints [136.12, -12.924, 22.115, -98.732, 46.823, 116.742, 25, 61.878]
  MoveL 202 to (85.97, 45.07, 115.69) mm, rotated rx 140.93 ry 0 rz -62.03 deg; joints [136.126, -12.916, 22.106, -98.73, 46.829, 116.719, 25, 62.03]
  MoveL 203 to (86.13, 44.14, 115.93) mm, rotated rx 140.93 ry 0 rz -62.03 deg; joints [136.157, -12.932, 22.116, -98.714, 46.859, 116.705, 25, 62.03]
  MoveL 204 to (86.12, 43.12, 116.32) mm, rotated rx 141.16 ry 0 rz -62.56 deg; joints [136.224, -12.842, 22.017, -98.687, 46.923, 116.45, 25, 62.563]
  MoveL 205 to (86.12, 43.1, 116.33) mm, rotated rx 141.3 ry 0 rz -63.76 deg; joints [136.206, -12.733, 21.915, -98.698, 46.906, 116.321, 25, 63.761]
  MoveL 206 to (86.62, 42.44, 116.21) mm, rotated rx 141.23 ry 0 rz -64.25 deg; joints [136.185, -12.762, 21.947, -98.707, 46.886, 116.402, 25, 64.245]
  MoveL 207 to (86.79, 42.19, 116.17) mm, rotated rx 141.23 ry 0 rz -64.25 deg; joints [136.192, -12.773, 21.957, -98.704, 46.892, 116.398, 25, 64.245]
  MoveL 208 to (87.08, 41.69, 116.13) mm, rotated rx 141.2 ry 0 rz -64.58 deg; joints [136.185, -12.783, 21.967, -98.707, 46.885, 116.425, 25, 64.583]
  MoveL 209 to (87.25, 41.36, 116.12) mm, rotated rx 141.2 ry 0 rz -64.58 deg; joints [136.194, -12.795, 21.977, -98.702, 46.894, 116.421, 25, 64.583]
  MoveL 210 to (89.56, 35.65, 116.25) mm, rotated rx 141.28 ry 0 rz -68.24 deg; joints [136.216, -12.764, 21.944, -98.693, 46.915, 116.335, 25, 68.243]
  MoveL 211 to (89.72, 35.04, 116.32) mm, rotated rx 141.28 ry 0 rz -68.24 deg; joints [136.234, -12.781, 21.957, -98.684, 46.932, 116.326, 25, 68.243]
  MoveL 212 to (89.79, 34.57, 116.4) mm, rotated rx 141.33 ry 0 rz -68.52 deg; joints [136.249, -12.761, 21.934, -98.678, 46.947, 116.268, 25, 68.523]
  MoveL 213 to (89.82, 34.13, 116.51) mm, rotated rx 141.33 ry 0 rz -68.52 deg; joints [136.264, -12.769, 21.939, -98.671, 46.961, 116.261, 25, 68.523]
  MoveL 214 to (89.71, 29.88, 117.75) mm, rotated rx 142.08 ry 0 rz -70.88 deg; joints [136.48, -12.471, 21.617, -98.583, 47.168, 115.437, 25, 70.883]
  MoveL 215 to (89.69, 29.72, 117.82) mm, rotated rx 142.2 ry 0 rz -71.32 deg; joints [136.495, -12.414, 21.559, -98.579, 47.182, 115.318, 25, 71.323]
  MoveL 216 to (90.3, 24.27, 118.59) mm, rotated rx 142.67 ry 0 rz -74.6 deg; joints [136.631, -12.225, 21.357, -98.526, 47.313, 114.801, 25, 74.603]
  MoveL 217 to (90.61, 17.61, 119.53) mm, rotated rx 143.25 ry 0 rz -78.64 deg; joints [136.797, -11.992, 21.109, -98.463, 47.473, 114.167, 25, 78.639]
  MoveL 218 to (90.33, 16.36, 119.92) mm, rotated rx 143.25 ry 0 rz -78.64 deg; joints [136.842, -12.008, 21.117, -98.444, 47.516, 114.148, 25, 78.639]
  MoveL 219 to (89.52, 15.51, 120.64) mm, rotated rx 143.25 ry 0 rz -78.64 deg; joints [136.887, -11.99, 21.094, -98.426, 47.559, 114.132, 25, 78.639]
  MoveL 220 to (88.71, 15.31, 121.26) mm, rotated rx 143.25 ry 0 rz -78.64 deg; joints [136.911, -11.957, 21.058, -98.416, 47.583, 114.124, 25, 78.639]
  MoveL 221 to (87.75, 15.63, 121.92) mm, rotated rx 143.25 ry 0 rz -78.64 deg; joints [136.924, -11.906, 21.007, -98.413, 47.595, 114.122, 25, 78.639]
  MoveL 222 to (87.03, 16.36, 122.33) mm, rotated rx 143.25 ry 0 rz -78.64 deg; joints [136.919, -11.856, 20.961, -98.418, 47.59, 114.127, 25, 78.639]
  MoveL 223 to (86.62, 17.37, 122.48) mm, rotated rx 143.25 ry 0 rz -78.64 deg; joints [136.897, -11.814, 20.924, -98.428, 47.57, 114.138, 25, 78.639]
  MoveL 224 to (85.75, 21.09, 122.51) mm, rotated rx 143.27 ry 0 rz -76.16 deg; joints [136.903, -11.807, 20.916, -98.427, 47.575, 114.118, 25, 76.164]
  MoveL 225 to (84.62, 25.11, 122.54) mm, rotated rx 143.29 ry 0 rz -73.45 deg; joints [136.908, -11.799, 20.908, -98.425, 47.581, 114.097, 25, 73.454]
  MoveL 226 to (84.64, 25.05, 122.54) mm, rotated rx 143.41 ry 0 rz -72.71 deg; joints [136.967, -11.797, 20.898, -98.4, 47.637, 113.949, 25, 72.708]
  MoveL 227 to (82.86, 26.95, 123.35) mm, rotated rx 143.94 ry 0 rz -71.16 deg; joints [137.119, -11.582, 20.672, -98.346, 47.783, 113.373, 25, 71.155]
  MoveL 228 to (82.69, 27.15, 123.42) mm, rotated rx 143.94 ry 0 rz -71.16 deg; joints [137.116, -11.57, 20.661, -98.348, 47.78, 113.375, 25, 71.155]
  MoveL 229 to (82.43, 27.47, 123.52) mm, rotated rx 144.01 ry 0 rz -70.9 deg; joints [137.135, -11.543, 20.633, -98.342, 47.799, 113.303, 25, 70.9]
  MoveL 230 to (80.51, 29.65, 124.28) mm, rotated rx 144.53 ry 0 rz -69.06 deg; joints [137.283, -11.335, 20.416, -98.291, 47.943, 112.742, 25, 69.055]
  Set speed (16.7 mm/s)
  MoveL 231 to (91.35, 33.8, 140.57) mm, rotated rx 144.53 ry 0 rz -69.06 deg; joints [137.198, -11.482, 19.837, -97.664, 47.759, 111.789, 25, 69.055]
  Set speed (1000.0 mm/s)
  MoveL 232 to (87.3, 33, 143.31) mm, rotated rx 146.24 ry 0 rz -68.43 deg; joints [137.697, -10.778, 19.116, -97.517, 48.246, 109.97, 25, 68.426]
  Set speed (5.0 mm/s)
  MoveL 233 to (76.96, 28.91, 126.68) mm, rotated rx 146.24 ry 0 rz -68.43 deg; joints [137.767, -10.651, 19.713, -98.137, 48.413, 110.919, 25, 68.426]
  Set speed (16.7 mm/s)
  MoveL 234 to (74.45, 30.84, 127.73) mm, rotated rx 146.98 ry 0 rz -66.48 deg; joints [137.974, -10.345, 19.405, -98.077, 48.615, 110.136, 25, 66.482]
  MoveL 235 to (73.91, 31.36, 127.91) mm, rotated rx 146.98 ry 0 rz -66.48 deg; joints [137.964, -10.313, 19.375, -98.083, 48.605, 110.142, 25, 66.482]
  MoveL 236 to (73.69, 31.64, 127.97) mm, rotated rx 147.02 ry 0 rz -66.24 deg; joints [137.975, -10.296, 19.358, -98.079, 48.617, 110.099, 25, 66.238]
  MoveL 237 to (73.56, 31.82, 128) mm, rotated rx 147.02 ry 0 rz -66.24 deg; joints [137.971, -10.287, 19.351, -98.081, 48.613, 110.101, 25, 66.238]
  MoveL 238 to (71.61, 34.59, 128.39) mm, rotated rx 147.3 ry 0 rz -63.84 deg; joints [138.048, -10.172, 19.236, -98.06, 48.688, 109.808, 25, 63.842]
  MoveL 239 to (71.26, 35.29, 128.38) mm, rotated rx 148.41 ry 0 rz -61.88 deg; joints [138.339, -9.865, 18.924, -97.975, 48.972, 108.637, 25, 61.88]
  MoveL 240 to (70.59, 34.73, 128.91) mm, rotated rx 148.79 ry 0 rz -62.01 deg; joints [138.443, -9.707, 18.768, -97.948, 49.074, 108.241, 25, 62.014]
  MoveL 241 to (70.2, 34.48, 129.19) mm, rotated rx 148.79 ry 0 rz -62.01 deg; joints [138.456, -9.69, 18.751, -97.945, 49.087, 108.239, 25, 62.014]
  MoveL 242 to (69.17, 34.3, 129.79) mm, rotated rx 148.79 ry 0 rz -62.01 deg; joints [138.473, -9.64, 18.704, -97.942, 49.104, 108.239, 25, 62.014]
  MoveL 243 to (68.72, 34.35, 130.02) mm, rotated rx 148.96 ry 0 rz -61.83 deg; joints [138.519, -9.571, 18.636, -97.93, 49.149, 108.066, 25, 61.826]
  MoveL 244 to (68.28, 34.44, 130.23) mm, rotated rx 148.96 ry 0 rz -61.83 deg; joints [138.521, -9.548, 18.614, -97.931, 49.151, 108.067, 25, 61.826]
  MoveL 245 to (67.34, 35, 130.57) mm, rotated rx 148.96 ry 0 rz -61.83 deg; joints [138.512, -9.497, 18.568, -97.937, 49.143, 108.074, 25, 61.826]
  MoveL 246 to (64.99, 37.06, 131.19) mm, rotated rx 149.43 ry 0 rz -59.58 deg; joints [138.64, -9.3, 18.376, -97.906, 49.269, 107.587, 25, 59.575]
  MoveL 247 to (64.7, 37.38, 131.24) mm, rotated rx 149.48 ry 0 rz -59.23 deg; joints [138.654, -9.281, 18.358, -97.903, 49.282, 107.537, 25, 59.232]
  MoveL 248 to (62.31, 39.22, 131.86) mm, rotated rx 149.95 ry 0 rz -57.04 deg; joints [138.783, -9.081, 18.164, -97.873, 49.41, 107.046, 25, 57.039]
  MoveL 249 to (61.89, 39.47, 131.98) mm, rotated rx 150.04 ry 0 rz -56.76 deg; joints [138.805, -9.042, 18.127, -97.869, 49.431, 106.961, 25, 56.765]
  MoveL 250 to (59.39, 41.34, 132.56) mm, rotated rx 150.49 ry 0 rz -54.43 deg; joints [138.928, -8.85, 17.943, -97.842, 49.552, 106.492, 25, 54.432]
  MoveL 251 to (59.02, 41.65, 132.62) mm, rotated rx 150.53 ry 0 rz -54.16 deg; joints [138.935, -8.831, 17.925, -97.841, 49.559, 106.46, 25, 54.158]
  MoveL 252 to (56.54, 43.48, 133.11) mm, rotated rx 150.92 ry 0 rz -51.79 deg; joints [139.04, -8.665, 17.767, -97.819, 49.664, 106.058, 25, 51.791]
  MoveL 253 to (56.15, 43.82, 133.17) mm, rotated rx 150.92 ry 0 rz -51.79 deg; joints [139.03, -8.646, 17.75, -97.823, 49.654, 106.062, 25, 51.791]
  MoveL 254 to (55.97, 44, 133.19) mm, rotated rx 150.93 ry 0 rz -51.59 deg; joints [139.034, -8.641, 17.745, -97.823, 49.657, 106.05, 25, 51.589]
  MoveL 255 to (54.6, 45.38, 133.29) mm, rotated rx 151.01 ry 0 rz -50.05 deg; joints [139.055, -8.605, 17.711, -97.818, 49.679, 105.966, 25, 50.048]
  MoveL 256 to (52.84, 46.44, 133.63) mm, rotated rx 151.34 ry 0 rz -48 deg; joints [139.155, -8.486, 17.598, -97.795, 49.777, 105.625, 25, 48.003]
  MoveL 257 to (51.9, 47.35, 133.68) mm, rotated rx 151.34 ry 0 rz -48 deg; joints [139.125, -8.444, 17.56, -97.808, 49.748, 105.636, 25, 48.003]
  MoveL 258 to (51.82, 47.48, 133.67) mm, rotated rx 151.33 ry 0 rz -47.88 deg; joints [139.122, -8.449, 17.564, -97.808, 49.745, 105.647, 25, 47.877]
  MoveL 259 to (51.47, 48.26, 133.53) mm, rotated rx 151.33 ry 0 rz -47.88 deg; joints [139.095, -8.435, 17.553, -97.818, 49.719, 105.655, 25, 47.877]
  MoveL 260 to (51.2, 49.25, 133.27) mm, rotated rx 151.12 ry 0 rz -47.13 deg; joints [139.039, -8.524, 17.637, -97.829, 49.664, 105.869, 25, 47.128]
  MoveL 261 to (51.21, 49.21, 133.27) mm, rotated rx 151 ry 0 rz -46.29 deg; joints [139.04, -8.597, 17.704, -97.824, 49.664, 105.985, 25, 46.288]
  MoveL 262 to (50.57, 49.97, 133.24) mm, rotated rx 150.97 ry 0 rz -45.5 deg; joints [139.032, -8.609, 17.715, -97.825, 49.657, 106.013, 25, 45.495]
  MoveL 263 to (50.14, 50.63, 133.15) mm, rotated rx 150.97 ry 0 rz -45.5 deg; joints [139.009, -8.592, 17.701, -97.833, 49.634, 106.021, 25, 45.495]
  MoveL 264 to (49.96, 51.08, 133.05) mm, rotated rx 150.95 ry 0 rz -45.4 deg; joints [138.992, -8.596, 17.706, -97.839, 49.618, 106.044, 25, 45.398]
  MoveL 265 to (49.78, 51.65, 132.89) mm, rotated rx 150.83 ry 0 rz -44.97 deg; joints [138.959, -8.648, 17.755, -97.845, 49.585, 106.17, 25, 44.974]
  MoveL 266 to (49.8, 51.61, 132.9) mm, rotated rx 150.7 ry 0 rz -43.94 deg; joints [138.965, -8.732, 17.832, -97.838, 49.589, 106.292, 25, 43.942]
  MoveL 267 to (48.92, 52.42, 132.91) mm, rotated rx 150.71 ry 0 rz -42.99 deg; joints [138.967, -8.728, 17.829, -97.838, 49.592, 106.283, 25, 42.988]
  MoveL 268 to (48.42, 53.02, 132.86) mm, rotated rx 150.71 ry 0 rz -42.99 deg; joints [138.945, -8.708, 17.812, -97.846, 49.571, 106.29, 25, 42.988]
  MoveL 269 to (48.33, 53.17, 132.83) mm, rotated rx 150.69 ry 0 rz -42.85 deg; joints [138.94, -8.717, 17.82, -97.847, 49.565, 106.311, 25, 42.854]
  MoveL 270 to (48.11, 53.58, 132.75) mm, rotated rx 150.69 ry 0 rz -42.85 deg; joints [138.925, -8.71, 17.814, -97.852, 49.551, 106.315, 25, 42.854]
  MoveL 271 to (47.66, 54.65, 132.47) mm, rotated rx 150.47 ry 0 rz -42.02 deg; joints [138.867, -8.802, 17.902, -97.865, 49.493, 106.538, 25, 42.017]
  MoveL 272 to (47.68, 54.65, 132.47) mm, rotated rx 150.36 ry 0 rz -41.42 deg; joints [138.864, -8.86, 17.956, -97.862, 49.49, 106.636, 25, 41.415]
  MoveL 273 to (45.09, 57.02, 132.37) mm, rotated rx 150.28 ry 0 rz -38.45 deg; joints [138.847, -8.902, 17.996, -97.864, 49.474, 106.721, 25, 38.453]
  MoveL 274 to (44.64, 57.53, 132.31) mm, rotated rx 150.28 ry 0 rz -38.45 deg; joints [138.828, -8.887, 17.982, -97.872, 49.455, 106.727, 25, 38.453]
  MoveL 275 to (44.55, 57.65, 132.28) mm, rotated rx 150.26 ry 0 rz -38.34 deg; joints [138.823, -8.895, 17.99, -97.873, 49.45, 106.747, 25, 38.337]
  MoveL 276 to (44.4, 57.89, 132.23) mm, rotated rx 150.26 ry 0 rz -38.34 deg; joints [138.813, -8.891, 17.987, -97.876, 49.441, 106.75, 25, 38.337]
  MoveL 277 to (43.89, 58.79, 132) mm, rotated rx 150.08 ry 0 rz -37.58 deg; joints [138.765, -8.966, 18.06, -97.887, 49.393, 106.935, 25, 37.583]
  MoveL 278 to (43.93, 58.75, 132) mm, rotated rx 149.99 ry 0 rz -36.93 deg; joints [138.769, -9.023, 18.112, -97.882, 49.396, 107.018, 25, 36.93]
  MoveL 279 to (43.1, 59.45, 131.97) mm, rotated rx 149.96 ry 0 rz -36.08 deg; joints [138.761, -9.036, 18.124, -97.884, 49.388, 107.049, 25, 36.081]
  MoveL 280 to (42.55, 60.06, 131.87) mm, rotated rx 149.96 ry 0 rz -36.08 deg; joints [138.736, -9.018, 18.109, -97.893, 49.364, 107.057, 25, 36.081]
  MoveL 281 to (42.43, 60.25, 131.82) mm, rotated rx 149.93 ry 0 rz -35.92 deg; joints [138.727, -9.032, 18.123, -97.895, 49.355, 107.092, 25, 35.922]
  MoveL 282 to (42.18, 60.7, 131.69) mm, rotated rx 149.93 ry 0 rz -35.92 deg; joints [138.709, -9.027, 18.119, -97.901, 49.339, 107.097, 25, 35.922]
  MoveL 283 to (41.74, 61.75, 131.34) mm, rotated rx 149.66 ry 0 rz -35.16 deg; joints [138.637, -9.141, 18.229, -97.918, 49.267, 107.375, 25, 35.163]
  MoveL 284 to (41.74, 61.75, 131.34) mm, rotated rx 149.52 ry 0 rz -33.53 deg; joints [138.66, -9.252, 18.331, -97.903, 49.288, 107.499, 25, 33.529]
  MoveL 285 to (38.81, 62.72, 131.78) mm, rotated rx 149.85 ry 0 rz -31.21 deg; joints [138.752, -9.11, 18.193, -97.882, 49.379, 107.15, 25, 31.206]
  MoveL 286 to (38.37, 62.9, 131.83) mm, rotated rx 149.85 ry 0 rz -31.21 deg; joints [138.742, -9.093, 18.178, -97.886, 49.369, 107.154, 25, 31.206]
  MoveL 287 to (38.1, 63.04, 131.84) mm, rotated rx 149.87 ry 0 rz -30.97 deg; joints [138.745, -9.088, 18.173, -97.885, 49.372, 107.142, 25, 30.968]
  MoveL 288 to (35.74, 64.17, 131.95) mm, rotated rx 149.95 ry 0 rz -28.95 deg; joints [138.768, -9.051, 18.138, -97.88, 49.395, 107.053, 25, 28.951]
  MoveL 289 to (33.28, 64.63, 132.38) mm, rotated rx 150.33 ry 0 rz -26.6 deg; joints [138.883, -8.913, 18.004, -97.852, 49.508, 106.658, 25, 26.601]
  MoveL 290 to (32.52, 64.87, 132.44) mm, rotated rx 150.33 ry 0 rz -26.6 deg; joints [138.866, -8.885, 17.978, -97.859, 49.492, 106.665, 25, 26.601]
  MoveL 291 to (31.84, 65.29, 132.4) mm, rotated rx 150.44 ry 0 rz -25.01 deg; joints [138.917, -8.89, 17.981, -97.843, 49.542, 106.549, 25, 25.005]
  MoveL 292 to (31.04, 65.26, 132.61) mm, rotated rx 150.6 ry 0 rz -24.44 deg; joints [138.961, -8.821, 17.914, -97.833, 49.585, 106.381, 25, 24.438]
  Set speed (16.7 mm/s)
  MoveL 293 to (35.1, 74.19, 150.04) mm, rotated rx 150.6 ry 0 rz -24.44 deg; joints [138.928, -8.898, 17.27, -97.231, 49.458, 105.446, 25, 24.438]
  Set speed (1000.0 mm/s)
  MoveL 294 to (31.87, 77.18, 149.24) mm, rotated rx 149.94 ry 0 rz -22.56 deg; joints [138.716, -9.13, 17.496, -97.28, 49.249, 106.134, 25, 22.558]
  Set speed (5.0 mm/s)
  MoveL 295 to (28.02, 67.93, 131.93) mm, rotated rx 149.94 ry 0 rz -22.56 deg; joints [138.755, -9.045, 18.133, -97.885, 49.382, 107.072, 25, 22.558]
  Set speed (16.7 mm/s)
  MoveL 296 to (27.16, 68.34, 131.9) mm, rotated rx 149.91 ry 0 rz -21.81 deg; joints [138.747, -9.056, 18.144, -97.887, 49.375, 107.099, 25, 21.808]
  MoveL 297 to (26.15, 68.55, 132) mm, rotated rx 150 ry 0 rz -20.54 deg; joints [138.785, -9.039, 18.126, -97.876, 49.412, 107.004, 25, 20.542]
  Set speed (16.7 mm/s)
  MoveL 298 to (29.66, 77.92, 149.32) mm, rotated rx 150 ry 0 rz -20.54 deg; joints [138.747, -9.124, 17.488, -97.271, 49.279, 106.067, 25, 20.542]
  Set speed (1000.0 mm/s)
  MoveL 299 to (28.49, 75.29, 150.89) mm, rotated rx 151.46 ry 0 rz -19.25 deg; joints [139.169, -8.574, 16.961, -97.183, 49.696, 104.565, 25, 19.254]
  Set speed (5.0 mm/s)
  MoveL 300 to (25.34, 66.27, 133.32) mm, rotated rx 151.46 ry 0 rz -19.25 deg; joints [139.196, -8.507, 17.615, -97.782, 49.816, 105.498, 25, 19.254]
  Set speed (16.7 mm/s)
  MoveL 301 to (22.18, 64.04, 134.96) mm, rotated rx 152.84 ry 0 rz -17.33 deg; joints [139.56, -7.924, 17.069, -97.714, 50.178, 104.108, 25, 17.327]
  MoveL 302 to (21.45, 63.67, 135.25) mm, rotated rx 152.84 ry 0 rz -17.33 deg; joints [139.559, -7.885, 17.034, -97.717, 50.177, 104.112, 25, 17.327]
  MoveL 303 to (21.08, 63.56, 135.36) mm, rotated rx 152.93 ry 0 rz -17.05 deg; joints [139.584, -7.844, 16.995, -97.713, 50.202, 104.015, 25, 17.051]
  MoveL 304 to (17.76, 62.26, 136.44) mm, rotated rx 153.9 ry 0 rz -14.48 deg; joints [139.838, -7.435, 16.62, -97.672, 50.455, 103.045, 25, 14.481]
  MoveL 305 to (16.46, 62.07, 136.69) mm, rotated rx 153.9 ry 0 rz -14.48 deg; joints [139.82, -7.38, 16.57, -97.681, 50.438, 103.055, 25, 14.481]
  MoveL 306 to (16.13, 62.11, 136.71) mm, rotated rx 153.92 ry 0 rz -14.19 deg; joints [139.825, -7.371, 16.562, -97.68, 50.444, 103.034, 25, 14.194]
  MoveL 307 to (15.19, 62.37, 136.7) mm, rotated rx 153.92 ry 0 rz -14.19 deg; joints [139.8, -7.344, 16.537, -97.689, 50.42, 103.042, 25, 14.194]
  MoveL 308 to (12.24, 63.71, 136.37) mm, rotated rx 153.63 ry 0 rz -11.37 deg; joints [139.726, -7.467, 16.65, -97.701, 50.345, 103.329, 25, 11.367]
  MoveL 309 to (10.77, 64.05, 136.34) mm, rotated rx 153.58 ry 0 rz -9.67 deg; joints [139.724, -7.499, 16.679, -97.699, 50.343, 103.378, 25, 9.674]
  MoveL 310 to (9.59, 64.64, 136.15) mm, rotated rx 153.58 ry 0 rz -9.67 deg; joints [139.683, -7.477, 16.66, -97.712, 50.304, 103.388, 25, 9.674]
  MoveL 311 to (9.4, 64.8, 136.09) mm, rotated rx 153.52 ry 0 rz -9.48 deg; joints [139.668, -7.502, 16.682, -97.714, 50.289, 103.446, 25, 9.482]
  MoveL 312 to (8.95, 65.31, 135.87) mm, rotated rx 153.52 ry 0 rz -9.48 deg; joints [139.645, -7.503, 16.684, -97.721, 50.266, 103.45, 25, 9.482]
  MoveL 313 to (8.07, 66.63, 135.28) mm, rotated rx 153.01 ry 0 rz -8.54 deg; joints [139.512, -7.72, 16.885, -97.743, 50.134, 103.962, 25, 8.545]
  MoveL 314 to (8.08, 66.6, 135.3) mm, rotated rx 152.7 ry 0 rz -7.41 deg; joints [139.481, -7.865, 17.018, -97.741, 50.101, 104.265, 25, 7.406]
  MoveL 315 to (7.87, 66.7, 135.26) mm, rotated rx 152.65 ry 0 rz -6.63 deg; joints [139.485, -7.906, 17.055, -97.737, 50.105, 104.313, 25, 6.626]
  MoveL 316 to (6.44, 66.79, 135.3) mm, rotated rx 152.68 ry 0 rz -5.41 deg; joints [139.493, -7.894, 17.044, -97.736, 50.113, 104.285, 25, 5.411]
  MoveL 317 to (4.06, 66.43, 135.57) mm, rotated rx 152.94 ry 0 rz -2.9 deg; joints [139.575, -7.801, 16.956, -97.719, 50.194, 104.012, 25, 2.901]
  MoveL 318 to (3.18, 66.36, 135.62) mm, rotated rx 152.95 ry 0 rz -2.81 deg; joints [139.561, -7.77, 16.928, -97.725, 50.181, 104.007, 25, 2.813]
  MoveL 319 to (2.64, 66.4, 135.61) mm, rotated rx 152.95 ry 0 rz -2.35 deg; joints [139.559, -7.772, 16.931, -97.725, 50.179, 104.013, 25, 2.346]
  MoveL 320 to (2.34, 66.35, 135.64) mm, rotated rx 152.98 ry 0 rz -1.78 deg; joints [139.575, -7.771, 16.929, -97.721, 50.195, 103.981, 25, 1.784]
  MoveL 321 to (0.65, 66.22, 135.73) mm, rotated rx 153.05 ry 0 rz -0.32 deg; joints [139.595, -7.74, 16.901, -97.718, 50.214, 103.908, 25, 0.324]
  Set speed (16.7 mm/s)
  MoveL 322 to (0.7, 75.28, 153.55) mm, rotated rx 153.05 ry 0 rz -0.32 deg; joints [139.58, -7.789, 16.231, -97.126, 50.107, 102.981, 25, 0.324]
  Set speed (1000.0 mm/s)
  MoveL 323 to (0.38, 81.25, 150.48) mm, rotated rx 151.91 ry 0 rz -1.95 deg; joints [139.134, -8.322, 16.731, -97.211, 49.665, 104.152, 25, 1.952]
  Set speed (5.0 mm/s)
  MoveL 324 to (0.06, 71.84, 132.84) mm, rotated rx 151.91 ry 0 rz -1.95 deg; joints [139.157, -8.259, 17.389, -97.811, 49.781, 105.085, 25, 1.952]
  Set speed (16.7 mm/s)
  MoveL 325 to (0.46, 72.78, 132.32) mm, rotated rx 151.5 ry 0 rz -2.24 deg; joints [139.049, -8.431, 17.552, -97.832, 49.674, 105.497, 25, 2.236]
  MoveL 326 to (0.48, 72.81, 132.3) mm, rotated rx 150.69 ry 0 rz -2.06 deg; joints [138.882, -8.71, 17.817, -97.866, 49.51, 106.322, 25, 2.06]
  MoveL 327 to (-0.2, 73.83, 131.74) mm, rotated rx 150.24 ry 0 rz -1.5 deg; joints [138.762, -8.899, 17.997, -97.892, 49.391, 106.781, 25, 1.499]
  MoveL 328 to (-0.16, 73.8, 131.76) mm, rotated rx 149.91 ry 0 rz 1.02 deg; joints [138.773, -9.108, 18.19, -97.875, 49.4, 107.092, 25, -1.021]
  MoveL 329 to (-0.94, 73.43, 131.96) mm, rotated rx 150.07 ry 0 rz 1.63 deg; joints [138.817, -9.04, 18.125, -97.865, 49.442, 106.927, 25, -1.634]
  MoveL 330 to (-1, 73.35, 132.01) mm, rotated rx 151.44 ry 0 rz 2.45 deg; joints [139.134, -8.61, 17.712, -97.794, 49.755, 105.522, 25, -2.454]
  MoveL 331 to (0.11, 71.82, 132.84) mm, rotated rx 152.1 ry 0 rz 1.62 deg; joints [139.309, -8.33, 17.449, -97.759, 49.929, 104.855, 25, -1.622]
  Set speed (16.7 mm/s)
  MoveL 332 to (-0.15, 81.18, 150.52) mm, rotated rx 152.1 ry 0 rz 1.62 deg; joints [139.288, -8.391, 16.788, -97.163, 49.814, 103.925, 25, -1.622]
  Set speed (1000.0 mm/s)
  MoveL 333 to (-2.2, 76.44, 152.97) mm, rotated rx 152.72 ry 0 rz 2.61 deg; joints [139.51, -7.974, 16.401, -97.132, 50.036, 103.301, 25, -2.613]
  Set speed (5.0 mm/s)
  MoveL 334 to (-1.78, 67.29, 135.19) mm, rotated rx 152.72 ry 0 rz 2.61 deg; joints [139.527, -7.921, 17.067, -97.724, 50.145, 104.228, 25, -2.613]
  Set speed (16.7 mm/s)
  MoveL 335 to (-4.6, 65.51, 136) mm, rotated rx 153.42 ry 0 rz 5.16 deg; joints [139.71, -7.623, 16.792, -97.693, 50.328, 103.526, 25, -5.157]
  MoveL 336 to (-5.37, 65.15, 136.14) mm, rotated rx 153.42 ry 0 rz 5.16 deg; joints [139.697, -7.589, 16.761, -97.7, 50.316, 103.533, 25, -5.157]
  MoveL 337 to (-5.53, 65.11, 136.15) mm, rotated rx 153.43 ry 0 rz 5.3 deg; joints [139.701, -7.583, 16.756, -97.699, 50.319, 103.519, 25, -5.298]
  MoveL 338 to (-6.84, 65.06, 136.12) mm, rotated rx 153.43 ry 0 rz 5.3 deg; joints [139.666, -7.547, 16.724, -97.711, 50.286, 103.53, 25, -5.298]
  MoveL 339 to (-8.18, 65.32, 135.92) mm, rotated rx 153.26 ry 0 rz 6.44 deg; joints [139.621, -7.621, 16.792, -97.719, 50.241, 103.703, 25, -6.442]
  MoveL 340 to (-8.39, 65.37, 135.88) mm, rotated rx 153.35 ry 0 rz 8.57 deg; joints [139.694, -7.659, 16.825, -97.695, 50.312, 103.592, 25, -8.575]
  MoveL 341 to (-8.78, 65.04, 136.01) mm, rotated rx 153.47 ry 0 rz 8.95 deg; joints [139.726, -7.608, 16.778, -97.69, 50.343, 103.472, 25, -8.946]
  MoveL 342 to (-9.88, 63.93, 136.46) mm, rotated rx 153.9 ry 0 rz 10.16 deg; joints [139.838, -7.431, 16.616, -97.672, 50.455, 103.046, 25, -10.164]
  MoveL 343 to (-10.85, 63.27, 136.7) mm, rotated rx 153.9 ry 0 rz 10.2 deg; joints [139.823, -7.384, 16.573, -97.68, 50.441, 103.057, 25, -10.196]
  MoveL 344 to (-11.5, 63.12, 136.72) mm, rotated rx 153.9 ry 0 rz 10.21 deg; joints [139.807, -7.364, 16.555, -97.686, 50.426, 103.064, 25, -10.213]
  MoveL 345 to (-12.33, 63.14, 136.63) mm, rotated rx 153.89 ry 0 rz 10.23 deg; joints [139.783, -7.348, 16.541, -97.694, 50.402, 103.072, 25, -10.235]
  MoveL 346 to (-13.46, 63.61, 136.31) mm, rotated rx 153.89 ry 0 rz 10.27 deg; joints [139.742, -7.345, 16.539, -97.705, 50.363, 103.083, 25, -10.268]
  MoveL 347 to (-14.09, 64.07, 136.03) mm, rotated rx 153.48 ry 0 rz 11.15 deg; joints [139.656, -7.52, 16.699, -97.716, 50.277, 103.49, 25, -11.154]
  MoveL 348 to (-14.97, 64.39, 135.78) mm, rotated rx 153.26 ry 0 rz 11.86 deg; joints [139.599, -7.614, 16.786, -97.726, 50.22, 103.709, 25, -11.859]
  MoveL 349 to (-15.61, 64.77, 135.53) mm, rotated rx 153 ry 0 rz 14.6 deg; joints [139.598, -7.801, 16.956, -97.712, 50.216, 103.953, 25, -14.598]
  MoveL 350 to (-16.81, 63.7, 135.89) mm, rotated rx 153.32 ry 0 rz 15.86 deg; joints [139.682, -7.665, 16.831, -97.698, 50.3, 103.633, 25, -15.855]
  MoveL 351 to (-17.27, 63.36, 135.99) mm, rotated rx 153.32 ry 0 rz 15.86 deg; joints [139.673, -7.642, 16.809, -97.702, 50.292, 103.637, 25, -15.855]
  MoveL 352 to (-18.51, 62.98, 136.01) mm, rotated rx 153.32 ry 0 rz 15.86 deg; joints [139.641, -7.602, 16.775, -97.714, 50.261, 103.648, 25, -15.855]
  MoveL 353 to (-19.16, 62.99, 135.91) mm, rotated rx 153.3 ry 0 rz 15.96 deg; joints [139.622, -7.599, 16.771, -97.72, 50.242, 103.664, 25, -15.957]
  MoveL 354 to (-19.83, 63.08, 135.77) mm, rotated rx 153.18 ry 0 rz 16.5 deg; joints [139.591, -7.65, 16.819, -97.725, 50.211, 103.784, 25, -16.499]
  MoveL 355 to (-19.77, 63.08, 135.78) mm, rotated rx 153.09 ry 0 rz 17.42 deg; joints [139.599, -7.714, 16.877, -97.718, 50.219, 103.869, 25, -17.42]
  MoveL 356 to (-22.31, 62.21, 135.79) mm, rotated rx 153.1 ry 0 rz 19.75 deg; joints [139.602, -7.71, 16.874, -97.718, 50.221, 103.86, 25, -19.747]
  MoveL 357 to (-23.19, 61.68, 135.89) mm, rotated rx 153.18 ry 0 rz 20.55 deg; joints [139.621, -7.672, 16.839, -97.715, 50.241, 103.777, 25, -20.548]
  MoveL 358 to (-25.79, 60.71, 135.86) mm, rotated rx 153.16 ry 0 rz 22.97 deg; joints [139.614, -7.684, 16.849, -97.716, 50.234, 103.804, 25, -22.969]
  MoveL 359 to (-26.87, 60.51, 135.74) mm, rotated rx 153.16 ry 0 rz 22.97 deg; joints [139.582, -7.662, 16.83, -97.727, 50.203, 103.813, 25, -22.969]
  MoveL 360 to (-27.89, 60.75, 135.42) mm, rotated rx 153.16 ry 0 rz 22.97 deg; joints [139.546, -7.661, 16.83, -97.737, 50.168, 103.82, 25, -22.969]
  MoveL 361 to (-28.22, 60.91, 135.28) mm, rotated rx 153.03 ry 0 rz 23.18 deg; joints [139.515, -7.713, 16.878, -97.743, 50.136, 103.942, 25, -23.179]
  MoveL 362 to (-28.59, 61.14, 135.1) mm, rotated rx 153.03 ry 0 rz 23.18 deg; joints [139.5, -7.719, 16.884, -97.747, 50.122, 103.944, 25, -23.179]
  MoveL 363 to (-30.65, 62.62, 133.96) mm, rotated rx 152.07 ry 0 rz 24.26 deg; joints [139.246, -8.128, 17.265, -97.793, 49.87, 104.916, 25, -24.259]
  MoveL 364 to (-31.61, 62.45, 133.82) mm, rotated rx 151.56 ry 0 rz 25.88 deg; joints [139.158, -8.341, 17.464, -97.804, 49.782, 105.426, 25, -25.879]
  MoveL 365 to (-32.47, 62.54, 133.57) mm, rotated rx 151.53 ry 0 rz 25.98 deg; joints [139.126, -8.349, 17.472, -97.814, 49.75, 105.457, 25, -25.975]
  MoveL 366 to (-33.8, 62.92, 133.06) mm, rotated rx 151.12 ry 0 rz 26.81 deg; joints [139.016, -8.524, 17.638, -97.836, 49.641, 105.879, 25, -26.806]
  MoveL 367 to (-34, 62.93, 133.01) mm, rotated rx 151.03 ry 0 rz 27.04 deg; joints [138.997, -8.562, 17.674, -97.839, 49.623, 105.969, 25, -27.039]
  MoveL 368 to (-35.34, 63.18, 132.54) mm, rotated rx 150.65 ry 0 rz 27.9 deg; joints [138.896, -8.721, 17.825, -97.861, 49.523, 106.354, 25, -27.904]
  MoveL 369 to (-35.85, 63.33, 132.33) mm, rotated rx 150.65 ry 0 rz 27.9 deg; joints [138.878, -8.724, 17.829, -97.866, 49.505, 106.358, 25, -27.904]
  MoveL 370 to (-36.74, 64.05, 131.74) mm, rotated rx 150.65 ry 0 rz 27.9 deg; joints [138.84, -8.751, 17.857, -97.876, 49.468, 106.364, 25, -27.904]
  MoveL 371 to (-36.85, 64.2, 131.64) mm, rotated rx 150.57 ry 0 rz 27.92 deg; joints [138.819, -8.785, 17.889, -97.881, 49.447, 106.447, 25, -27.92]
  MoveL 372 to (-37.14, 64.9, 131.21) mm, rotated rx 150.57 ry 0 rz 27.92 deg; joints [138.801, -8.817, 17.92, -97.885, 49.43, 106.448, 25, -27.92]
  MoveL 373 to (-37.3, 65.85, 130.69) mm, rotated rx 149.85 ry 0 rz 27.64 deg; joints [138.623, -9.09, 18.183, -97.926, 49.254, 107.193, 25, -27.642]
  MoveL 374 to (-37.74, 66.5, 130.23) mm, rotated rx 149.5 ry 0 rz 27.71 deg; joints [138.53, -9.234, 18.323, -97.948, 49.162, 107.547, 25, -27.708]
  MoveL 375 to (-37.7, 66.48, 130.25) mm, rotated rx 148.81 ry 0 rz 28.53 deg; joints [138.409, -9.497, 18.576, -97.972, 49.043, 108.253, 25, -28.532]
  MoveL 376 to (-39.22, 66.48, 129.81) mm, rotated rx 148.47 ry 0 rz 29.53 deg; joints [138.316, -9.639, 18.714, -97.996, 48.952, 108.604, 25, -29.531]
  MoveL 377 to (-39.52, 66.48, 129.71) mm, rotated rx 148.41 ry 0 rz 29.7 deg; joints [138.299, -9.663, 18.739, -98, 48.935, 108.666, 25, -29.7]
  MoveL 378 to (-40.34, 66.62, 129.39) mm, rotated rx 148.41 ry 0 rz 29.7 deg; joints [138.269, -9.664, 18.742, -98.011, 48.906, 108.674, 25, -29.7]
  MoveL 379 to (-43.07, 67.55, 128.02) mm, rotated rx 147.41 ry 0 rz 31.09 deg; joints [137.993, -10.082, 19.157, -98.085, 48.636, 109.726, 25, -31.09]
  MoveL 380 to (-43.88, 68.03, 127.49) mm, rotated rx 147.41 ry 0 rz 31.09 deg; joints [137.96, -10.102, 19.178, -98.096, 48.604, 109.735, 25, -31.09]
  MoveL 381 to (-44.34, 68.82, 126.91) mm, rotated rx 147.41 ry 0 rz 31.09 deg; joints [137.936, -10.138, 19.215, -98.102, 48.58, 109.739, 25, -31.09]
  MoveL 382 to (-44.39, 69.01, 126.79) mm, rotated rx 147.32 ry 0 rz 31.05 deg; joints [137.913, -10.173, 19.25, -98.109, 48.557, 109.828, 25, -31.053]
  MoveL 383 to (-44.37, 70.12, 126.18) mm, rotated rx 147.32 ry 0 rz 31.05 deg; joints [137.902, -10.229, 19.303, -98.11, 48.547, 109.826, 25, -31.053]
  MoveL 384 to (-43.57, 72.61, 125.05) mm, rotated rx 146.55 ry 0 rz 29.74 deg; joints [137.689, -10.547, 19.624, -98.172, 48.338, 110.638, 25, -29.736]
  MoveL 385 to (-43.37, 73.06, 124.86) mm, rotated rx 146.55 ry 0 rz 29.74 deg; joints [137.691, -10.571, 19.646, -98.17, 48.34, 110.636, 25, -29.736]
  MoveL 386 to (-43.28, 73.2, 124.8) mm, rotated rx 146.52 ry 0 rz 29.64 deg; joints [137.681, -10.586, 19.661, -98.173, 48.331, 110.674, 25, -29.641]
  MoveL 387 to (-43.07, 73.5, 124.7) mm, rotated rx 146.52 ry 0 rz 29.64 deg; joints [137.685, -10.603, 19.677, -98.171, 48.334, 110.671, 25, -29.641]
  MoveL 388 to (-41.36, 75.58, 124.03) mm, rotated rx 146.07 ry 0 rz 27.98 deg; joints [137.561, -10.785, 19.862, -98.209, 48.214, 111.141, 25, -27.977]
  MoveL 389 to (-40.95, 77.64, 122.89) mm, rotated rx 145.02 ry 0 rz 26.48 deg; joints [137.259, -11.158, 20.252, -98.309, 47.921, 112.27, 25, -26.477]
  MoveL 390 to (-40.13, 80.53, 121.29) mm, rotated rx 144 ry 0 rz 25.2 deg; joints [136.968, -11.576, 20.687, -98.409, 47.639, 113.376, 25, -25.2]
  Set speed (16.7 mm/s)
  MoveL 391 to (-45.13, 91.17, 137.47) mm, rotated rx 144 ry 0 rz 25.2 deg; joints [136.878, -11.73, 20.115, -97.776, 47.449, 112.419, 25, -25.2]
  Set speed (1000.0 mm/s)
  MoveL 392 to (-40.64, 95.64, 135.82) mm, rotated rx 143.37 ry 0 rz 23.46 deg; joints [136.745, -12.106, 20.492, -97.813, 47.318, 113.068, 25, -23.459]
  Set speed (5.0 mm/s)
  MoveL 393 to (-35.89, 84.7, 119.77) mm, rotated rx 143.37 ry 0 rz 23.46 deg; joints [136.84, -11.946, 21.058, -98.447, 47.514, 114.026, 25, -23.459]
  Set speed (16.7 mm/s)
  MoveL 394 to (-31.63, 85.22, 120.6) mm, rotated rx 143.89 ry 0 rz 20.87 deg; joints [136.988, -11.737, 20.838, -98.394, 47.657, 113.466, 25, -20.867]
  MoveL 395 to (-31.47, 85.24, 120.63) mm, rotated rx 143.91 ry 0 rz 20.77 deg; joints [136.993, -11.73, 20.83, -98.392, 47.662, 113.445, 25, -20.77]
  MoveL 396 to (-31.25, 85.28, 120.66) mm, rotated rx 143.95 ry 0 rz 20.52 deg; joints [136.999, -11.71, 20.811, -98.39, 47.668, 113.406, 25, -20.52]
  Set speed (16.7 mm/s)
  MoveL 397 to (-35.37, 96.3, 136.83) mm, rotated rx 143.95 ry 0 rz 20.52 deg; joints [136.909, -11.864, 20.238, -97.758, 47.477, 112.448, 25, -20.52]
  Set speed (1000.0 mm/s)
  MoveL 398 to (-28.57, 94.12, 139.9) mm, rotated rx 145.73 ry 0 rz 16.86 deg; joints [137.41, -11.1, 19.45, -97.604, 47.966, 110.547, 25, -16.855]
  Set speed (5.0 mm/s)
  MoveL 399 to (-25.31, 83.34, 123.38) mm, rotated rx 145.73 ry 0 rz 16.86 deg; joints [137.484, -10.966, 20.042, -98.229, 48.138, 111.499, 25, -16.855]
  Set speed (16.7 mm/s)
  MoveL 400 to (-22.08, 84.31, 123.33) mm, rotated rx 145.7 ry 0 rz 14.64 deg; joints [137.476, -10.977, 20.054, -98.232, 48.131, 111.528, 25, -14.636]
  MoveL 401 to (-20.8, 84.38, 123.51) mm, rotated rx 145.7 ry 0 rz 14.64 deg; joints [137.515, -11.006, 20.076, -98.215, 48.168, 111.513, 25, -14.636]
  MoveL 402 to (-19.95, 84.08, 123.85) mm, rotated rx 145.7 ry 0 rz 14.64 deg; joints [137.548, -11.009, 20.075, -98.203, 48.199, 111.501, 25, -14.636]
  MoveL 403 to (-19.21, 83.3, 124.5) mm, rotated rx 145.7 ry 0 rz 14.64 deg; joints [137.587, -10.987, 20.05, -98.189, 48.237, 111.49, 25, -14.636]
  MoveL 404 to (-19.04, 82.27, 125.2) mm, rotated rx 145.7 ry 0 rz 14.64 deg; joints [137.613, -10.943, 20.005, -98.181, 48.262, 111.484, 25, -14.636]
  MoveL 405 to (-19.14, 81.57, 125.65) mm, rotated rx 146.01 ry 0 rz 14.82 deg; joints [137.698, -10.817, 19.877, -98.155, 48.345, 111.159, 25, -14.823]
  MoveL 406 to (-19.61, 80.53, 126.25) mm, rotated rx 146.01 ry 0 rz 14.82 deg; joints [137.704, -10.759, 19.822, -98.155, 48.352, 111.162, 25, -14.823]
  MoveL 407 to (-20.6, 79.78, 126.57) mm, rotated rx 146.01 ry 0 rz 14.82 deg; joints [137.688, -10.705, 19.772, -98.164, 48.337, 111.171, 25, -14.823]
  MoveL 408 to (-24.91, 77.66, 127.1) mm, rotated rx 146.38 ry 0 rz 18.13 deg; joints [137.793, -10.55, 19.616, -98.133, 48.439, 110.774, 25, -18.133]
  MoveL 409 to (-24.9, 77.68, 127.09) mm, rotated rx 146.75 ry 0 rz 19.18 deg; joints [137.912, -10.477, 19.535, -98.093, 48.554, 110.374, 25, -19.182]
  MoveL 410 to (-25.42, 76.36, 127.79) mm, rotated rx 147.25 ry 0 rz 19.85 deg; joints [138.049, -10.272, 19.329, -98.054, 48.688, 109.852, 25, -19.852]
  MoveL 411 to (-25.89, 75.63, 128.13) mm, rotated rx 147.41 ry 0 rz 20.22 deg; joints [138.094, -10.193, 19.251, -98.042, 48.733, 109.684, 25, -20.219]
  MoveL 412 to (-26.43, 74.54, 128.65) mm, rotated rx 147.79 ry 0 rz 20.87 deg; joints [138.2, -10.034, 19.093, -98.013, 48.836, 109.283, 25, -20.865]
  MoveL 413 to (-25.86, 74.27, 128.93) mm, rotated rx 149.16 ry 0 rz 20.71 deg; joints [138.513, -9.573, 18.639, -97.932, 49.143, 107.868, 25, -20.71]
  MoveL 414 to (-24.57, 73.46, 129.64) mm, rotated rx 149.67 ry 0 rz 20.04 deg; joints [138.654, -9.357, 18.428, -97.898, 49.281, 107.335, 25, -20.039]
  MoveL 415 to (-24.22, 73.63, 129.61) mm, rotated rx 150.07 ry 0 rz 18.09 deg; joints [138.681, -9.161, 18.245, -97.902, 49.309, 106.951, 25, -18.089]
  MoveL 416 to (-23.88, 73.76, 129.6) mm, rotated rx 150.06 ry 0 rz 17.82 deg; joints [138.678, -9.165, 18.248, -97.902, 49.307, 106.959, 25, -17.824]
  MoveL 417 to (-22.47, 74.19, 129.6) mm, rotated rx 150.06 ry 0 rz 16.86 deg; joints [138.684, -9.169, 18.252, -97.901, 49.312, 106.954, 25, -16.858]
  MoveL 418 to (-22.37, 74.86, 129.24) mm, rotated rx 149.32 ry 0 rz 15.04 deg; joints [138.455, -9.37, 18.454, -97.964, 49.089, 107.737, 25, -15.043]
  MoveL 419 to (-22.31, 75.05, 129.14) mm, rotated rx 149.25 ry 0 rz 14.96 deg; joints [138.436, -9.4, 18.483, -97.969, 49.07, 107.811, 25, -14.963]
  MoveL 420 to (-22.08, 75.53, 128.9) mm, rotated rx 149.25 ry 0 rz 14.96 deg; joints [138.434, -9.427, 18.508, -97.968, 49.068, 107.809, 25, -14.963]
  MoveL 421 to (-21.38, 76.61, 128.38) mm, rotated rx 148.88 ry 0 rz 14.29 deg; joints [138.332, -9.584, 18.662, -97.994, 48.967, 108.198, 25, -14.285]
  MoveL 422 to (-21.39, 76.6, 128.38) mm, rotated rx 148.51 ry 0 rz 13.88 deg; joints [138.238, -9.686, 18.765, -98.02, 48.876, 108.583, 25, -13.881]
  MoveL 423 to (-21.22, 78.23, 127.43) mm, rotated rx 147.83 ry 0 rz 13.48 deg; joints [138.052, -9.968, 19.045, -98.07, 48.693, 109.292, 25, -13.485]
  MoveL 424 to (-20.87, 79.14, 126.92) mm, rotated rx 147.83 ry 0 rz 13.48 deg; joints [138.044, -10.017, 19.091, -98.07, 48.685, 109.29, 25, -13.485]
  MoveL 425 to (-20.67, 79.44, 126.76) mm, rotated rx 147.72 ry 0 rz 13.3 deg; joints [138.014, -10.062, 19.136, -98.078, 48.656, 109.402, 25, -13.3]
  MoveL 426 to (-19.98, 80.12, 126.45) mm, rotated rx 147.72 ry 0 rz 13.3 deg; joints [138.022, -10.107, 19.177, -98.073, 48.663, 109.396, 25, -13.3]
  MoveL 427 to (-17.08, 81.97, 125.69) mm, rotated rx 147.2 ry 0 rz 11.08 deg; joints [137.877, -10.324, 19.395, -98.114, 48.522, 109.946, 25, -11.084]
  MoveL 428 to (-17.09, 81.98, 125.67) mm, rotated rx 145.8 ry 0 rz 10.36 deg; joints [137.542, -10.746, 19.828, -98.218, 48.195, 111.428, 25, -10.362]
  MoveL 429 to (-18.66, 83.27, 124.6) mm, rotated rx 145.06 ry 0 rz 11.25 deg; joints [137.336, -11.047, 20.136, -98.284, 47.995, 112.211, 25, -11.252]
  Set speed (16.7 mm/s)
  MoveL 430 to (-20.89, 94.5, 141) mm, rotated rx 145.06 ry 0 rz 11.25 deg; joints [137.256, -11.188, 19.552, -97.657, 47.816, 111.258, 25, -11.252]
  Set speed (1000.0 mm/s)
  MoveL 431 to (-18.77, 98.7, 138.4) mm, rotated rx 144.84 ry 0 rz 11.08 deg; joints [137.168, -11.489, 19.848, -97.675, 47.73, 111.488, 25, -11.077]
  Set speed (5.0 mm/s)
  MoveL 432 to (-16.55, 87.4, 122.05) mm, rotated rx 144.84 ry 0 rz 11.08 deg; joints [137.25, -11.346, 20.43, -98.304, 47.911, 112.443, 25, -11.077]
  Set speed (16.7 mm/s)
  MoveL 433 to (-13.72, 87.38, 122.4) mm, rotated rx 145.07 ry 0 rz 9.28 deg; joints [137.316, -11.252, 20.333, -98.282, 47.974, 112.195, 25, -9.281]
  MoveL 434 to (-13.64, 87.42, 122.39) mm, rotated rx 145.08 ry 0 rz 8.65 deg; joints [137.294, -11.223, 20.308, -98.292, 47.954, 112.2, 25, -8.65]
  MoveL 435 to (-9.28, 88.48, 122.04) mm, rotated rx 144.85 ry 0 rz 5.77 deg; joints [137.229, -11.316, 20.405, -98.314, 47.891, 112.445, 25, -5.768]
  Set speed (16.7 mm/s)
  MoveL 436 to (-10.44, 99.93, 138.39) mm, rotated rx 144.85 ry 0 rz 5.77 deg; joints [137.147, -11.459, 19.822, -97.685, 47.71, 111.49, 25, -5.768]
  Set speed (1000.0 mm/s)
  MoveL 437 to (-7.68, 99.26, 139.05) mm, rotated rx 145.21 ry 0 rz 4.05 deg; joints [137.245, -11.297, 19.657, -97.655, 47.806, 111.109, 25, -4.052]
  Set speed (5.0 mm/s)
  MoveL 438 to (-6.88, 87.88, 122.63) mm, rotated rx 145.21 ry 0 rz 4.05 deg; joints [137.324, -11.158, 20.243, -98.283, 47.983, 112.063, 25, -4.052]
  Set speed (16.7 mm/s)
  MoveL 439 to (-6.64, 87.94, 122.59) mm, rotated rx 145.2 ry 0 rz 4 deg; joints [137.325, -11.168, 20.252, -98.282, 47.984, 112.07, 25, -4]
  MoveL 440 to (-5.17, 88.26, 122.44) mm, rotated rx 145.03 ry 0 rz 2.66 deg; joints [137.266, -11.213, 20.303, -98.303, 47.928, 112.259, 25, -2.659]
  MoveL 441 to (-2.33, 90.05, 121.22) mm, rotated rx 144.16 ry 0 rz 0.55 deg; joints [137.015, -11.548, 20.654, -98.391, 47.684, 113.202, 25, -0.553]
  MoveL 442 to (-1.85, 90.27, 121.06) mm, rotated rx 144.16 ry 0 rz 0.55 deg; joints [137.02, -11.572, 20.676, -98.387, 47.689, 113.198, 25, -0.553]
  MoveL 443 to (-1.69, 90.33, 121.02) mm, rotated rx 144.13 ry 0 rz 0.45 deg; joints [137.013, -11.582, 20.687, -98.39, 47.682, 113.226, 25, -0.451]
  MoveL 444 to (-1.28, 90.44, 120.94) mm, rotated rx 144.13 ry 0 rz 0.45 deg; joints [137.021, -11.6, 20.702, -98.386, 47.689, 113.222, 25, -0.451]
  MoveL 445 to (-0.56, 90.58, 120.84) mm, rotated rx 144.08 ry 0 rz 0 deg; joints [137.006, -11.621, 20.725, -98.391, 47.675, 113.277, 25, 0]
  MoveL 446 to (-0.09, 90.65, 120.79) mm, rotated rx 143.97 ry 0 rz -0.62 deg; joints [136.967, -11.642, 20.75, -98.407, 47.638, 113.398, 25, 0.621]
  MoveL 447 to (0.17, 90.74, 120.72) mm, rotated rx 143.93 ry 0 rz -0.78 deg; joints [136.954, -11.66, 20.769, -98.411, 47.625, 113.446, 25, 0.78]
  MoveL 448 to (3.8, 92.42, 119.38) mm, rotated rx 143.04 ry 0 rz -3.17 deg; joints [136.697, -12.006, 21.137, -98.506, 47.377, 114.415, 25, 3.17]
  MoveL 449 to (4.11, 92.58, 119.25) mm, rotated rx 142.93 ry 0 rz -3.43 deg; joints [136.664, -12.044, 21.179, -98.519, 47.346, 114.537, 25, 3.432]
  MoveL 450 to (7.34, 94.25, 117.77) mm, rotated rx 142 ry 0 rz -5.38 deg; joints [136.394, -12.412, 21.574, -98.624, 47.087, 115.561, 25, 5.382]
  MoveL 451 to (7.29, 94.23, 117.79) mm, rotated rx 141.72 ry 0 rz -5.75 deg; joints [136.315, -12.477, 21.65, -98.658, 47.011, 115.871, 25, 5.754]
  MoveL 452 to (8, 95.05, 117.08) mm, rotated rx 141.29 ry 0 rz -6.13 deg; joints [136.192, -12.646, 21.834, -98.708, 46.893, 116.341, 25, 6.126]
  MoveL 453 to (7.98, 95.04, 117.09) mm, rotated rx 140.27 ry 0 rz -5.99 deg; joints [135.963, -12.971, 22.189, -98.805, 46.674, 117.455, 25, 5.992]
  MoveL 454 to (7.61, 95.5, 116.74) mm, rotated rx 140.06 ry 0 rz -5.74 deg; joints [135.902, -13.053, 22.28, -98.832, 46.616, 117.688, 25, 5.744]
  Set speed (16.7 mm/s)
  MoveL 455 to (8.89, 108.27, 132.08) mm, rotated rx 140.06 ry 0 rz -5.74 deg; joints [135.776, -13.251, 21.751, -98.187, 46.385, 116.723, 25, 5.744]
  Set speed (1000.0 mm/s)
  MoveL 456 to (6.54, 110.49, 130.37) mm, rotated rx 139 ry 0 rz -4.16 deg; joints [135.48, -13.677, 22.221, -98.312, 46.102, 117.898, 25, 4.158]
  Set speed (5.0 mm/s)
  MoveL 457 to (5.59, 97.4, 115.28) mm, rotated rx 139 ry 0 rz -4.16 deg; joints [135.616, -13.467, 22.737, -98.959, 46.344, 118.865, 25, 4.158]
  Set speed (16.7 mm/s)
  MoveL 458 to (1.93, 99.67, 113.44) mm, rotated rx 137.93 ry 0 rz -1.95 deg; joints [135.301, -13.883, 23.208, -99.109, 46.046, 120.08, 25, 1.953]
  MoveL 459 to (-0.96, 100.61, 112.62) mm, rotated rx 137.37 ry 0 rz 0 deg; joints [135.156, -14.106, 23.458, -99.181, 45.908, 120.703, 25, 0]
  MoveL 460 to (-1.57, 100.68, 112.55) mm, rotated rx 137.27 ry 0 rz 0.5 deg; joints [135.136, -14.149, 23.504, -99.19, 45.89, 120.813, 25, -0.496]
  MoveL 461 to (-4.78, 101.28, 111.93) mm, rotated rx 136.92 ry 0 rz 2.31 deg; joints [135.031, -14.285, 23.661, -99.244, 45.791, 121.221, 25, -2.314]
  Set speed (16.7 mm/s)
  MoveL 462 to (-5.33, 114.93, 126.53) mm, rotated rx 136.92 ry 0 rz 2.31 deg; joints [134.874, -14.518, 23.169, -98.591, 45.525, 120.253, 25, -2.314]
  Set speed (1000.0 mm/s)
  MoveL 463 to (-6.43, 118.47, 123.16) mm, rotated rx 136.55 ry 0 rz 2.11 deg; joints [134.634, -14.734, 23.437, -98.713, 45.298, 120.743, 25, -2.11]
  Set speed (5.0 mm/s)
  MoveL 464 to (-5.93, 104.72, 108.65) mm, rotated rx 136.55 ry 0 rz 2.11 deg; joints [134.795, -14.497, 23.925, -99.369, 45.569, 121.714, 25, -2.11]
  Set speed (16.7 mm/s)
  MoveL 465 to (-5.24, 105.5, 107.92) mm, rotated rx 136.16 ry 0 rz 1.72 deg; joints [134.679, -14.644, 24.099, -99.431, 45.461, 122.166, 25, -1.723]
  MoveL 466 to (-5.14, 105.96, 107.49) mm, rotated rx 135.65 ry 0 rz 1.48 deg; joints [134.536, -14.803, 24.29, -99.51, 45.327, 122.753, 25, -1.478]
  MoveL 467 to (-4.87, 106.64, 106.81) mm, rotated rx 135.29 ry 0 rz 1.33 deg; joints [134.429, -14.937, 24.451, -99.571, 45.227, 123.173, 25, -1.328]
  MoveL 468 to (-4.79, 106.65, 106.82) mm, rotated rx 134.3 ry 0 rz 3.44 deg; joints [134.295, -15.364, 24.907, -99.644, 45.102, 124.24, 25, -3.44]
  MoveL 469 to (-5.42, 106.22, 107.21) mm, rotated rx 134.51 ry 0 rz 3.79 deg; joints [134.359, -15.285, 24.813, -99.607, 45.161, 123.991, 25, -3.79]
  MoveL 470 to (-5.39, 106.23, 107.2) mm, rotated rx 134.97 ry 0 rz 4.2 deg; joints [134.487, -15.177, 24.672, -99.534, 45.28, 123.458, 25, -4.199]
  MoveL 471 to (-5.89, 104.67, 108.71) mm, rotated rx 135.79 ry 0 rz 4.53 deg; joints [134.732, -14.869, 24.307, -99.398, 45.509, 122.502, 25, -4.534]
  Set speed (16.7 mm/s)
  MoveL 472 to (-6.99, 118.57, 123.04) mm, rotated rx 135.79 ry 0 rz 4.53 deg; joints [134.563, -15.115, 23.827, -98.743, 45.23, 121.532, 25, -4.534]
  Set speed (1000.0 mm/s)
  MoveL 473 to (-9.78, 115.15, 126.06) mm, rotated rx 136.65 ry 0 rz 4.89 deg; joints [134.814, -14.644, 23.306, -98.62, 45.468, 120.546, 25, -4.887]
  Set speed (5.0 mm/s)
  MoveL 474 to (-8.61, 101.47, 111.52) mm, rotated rx 136.65 ry 0 rz 4.89 deg; joints [134.973, -14.408, 23.796, -99.272, 45.736, 121.515, 25, -4.887]
  Set speed (16.7 mm/s)
  MoveL 475 to (-9.21, 101.41, 111.53) mm, rotated rx 136.66 ry 0 rz 5.23 deg; joints [134.975, -14.406, 23.793, -99.272, 45.738, 121.508, 25, -5.226]
  MoveL 476 to (-9.17, 101.41, 111.53) mm, rotated rx 136.98 ry 0 rz 6.22 deg; joints [135.098, -14.367, 23.726, -99.206, 45.853, 121.115, 25, -6.222]
  MoveL 477 to (-11.88, 98.43, 113.91) mm, rotated rx 138.36 ry 0 rz 7.98 deg; joints [135.503, -13.84, 23.123, -99.007, 46.236, 119.552, 25, -7.981]
  MoveL 478 to (-14.94, 94.64, 116.73) mm, rotated rx 140.02 ry 0 rz 10.12 deg; joints [135.993, -13.19, 22.395, -98.784, 46.701, 117.673, 25, -10.124]
  MoveL 479 to (-14.92, 94.66, 116.72) mm, rotated rx 140.72 ry 0 rz 10.45 deg; joints [136.166, -12.993, 22.173, -98.709, 46.866, 116.91, 25, -10.446]
  MoveL 480 to (-14.63, 93.76, 117.48) mm, rotated rx 141.18 ry 0 rz 10.37 deg; joints [136.299, -12.811, 21.974, -98.653, 46.993, 116.402, 25, -10.372]
  MoveL 481 to (-14.58, 93.06, 118.04) mm, rotated rx 141.18 ry 0 rz 10.37 deg; joints [136.318, -12.78, 21.941, -98.646, 47.012, 116.395, 25, -10.372]
  MoveL 482 to (-14.62, 92.8, 118.24) mm, rotated rx 141.3 ry 0 rz 10.42 deg; joints [136.353, -12.732, 21.889, -98.631, 47.046, 116.261, 25, -10.424]
  MoveL 483 to (-14.7, 92.49, 118.48) mm, rotated rx 141.3 ry 0 rz 10.42 deg; joints [136.359, -12.715, 21.872, -98.629, 47.051, 116.259, 25, -10.424]
  MoveL 484 to (-15.55, 89.92, 120.33) mm, rotated rx 142.45 ry 0 rz 11.25 deg; joints [136.692, -12.254, 21.375, -98.499, 47.371, 114.989, 25, -11.251]
  MoveL 485 to (-16.23, 88.97, 120.95) mm, rotated rx 142.7 ry 0 rz 11.66 deg; joints [136.766, -12.137, 21.251, -98.471, 47.443, 114.719, 25, -11.662]
  MoveL 486 to (-17.08, 87.31, 122.03) mm, rotated rx 143.4 ry 0 rz 12.42 deg; joints [136.967, -11.855, 20.953, -98.398, 47.636, 113.956, 25, -12.422]
  Set speed (16.7 mm/s)
  MoveL 487 to (-19.65, 98.95, 138.09) mm, rotated rx 143.4 ry 0 rz 12.42 deg; joints [136.872, -12.015, 20.386, -97.766, 47.441, 112.999, 25, -12.422]
  Set speed (1000.0 mm/s)
  MoveL 488 to (-23.25, 95.87, 139.7) mm, rotated rx 143.97 ry 0 rz 13.24 deg; joints [136.992, -11.658, 20.031, -97.735, 47.559, 112.415, 25, -13.245]
  Set speed (5.0 mm/s)
  MoveL 489 to (-20.56, 84.42, 123.52) mm, rotated rx 143.97 ry 0 rz 13.24 deg; joints [137.082, -11.505, 20.604, -98.365, 47.749, 113.371, 25, -13.245]
  Set speed (16.7 mm/s)
  MoveL 490 to (-23.6, 84.33, 123.04) mm, rotated rx 143.65 ry 0 rz 15.2 deg; joints [136.991, -11.634, 20.739, -98.397, 47.661, 113.716, 25, -15.201]
  MoveL 491 to (-23.58, 84.33, 123.04) mm, rotated rx 143.67 ry 0 rz 16.16 deg; joints [137.033, -11.674, 20.772, -98.378, 47.701, 113.678, 25, -16.155]
  MoveL 492 to (-24.36, 83.85, 123.22) mm, rotated rx 143.78 ry 0 rz 16.74 deg; joints [137.067, -11.626, 20.721, -98.366, 47.734, 113.549, 25, -16.736]
  Set speed (16.7 mm/s)
  MoveL 493 to (-27.76, 95.16, 139.36) mm, rotated rx 143.78 ry 0 rz 16.74 deg; joints [136.976, -11.782, 20.151, -97.736, 47.542, 112.593, 25, -16.736]
  Set speed (1000.0 mm/s)
  MoveL 494 to (-35.24, 96.75, 136.54) mm, rotated rx 142.35 ry 0 rz 19.11 deg; joints [136.479, -12.316, 20.733, -97.914, 47.062, 114.187, 25, -19.109]
  Set speed (5.0 mm/s)
  MoveL 495 to (-31.24, 85.21, 120.71) mm, rotated rx 142.35 ry 0 rz 19.11 deg; joints [136.583, -12.144, 21.287, -98.55, 47.268, 115.147, 25, -19.109]
  Set speed (16.7 mm/s)
  MoveL 496 to (-31.61, 85.31, 120.54) mm, rotated rx 142.24 ry 0 rz 19.31 deg; joints [136.553, -12.186, 21.332, -98.562, 47.239, 115.262, 25, -19.31]
  MoveL 497 to (-32.59, 85.86, 119.89) mm, rotated rx 142.24 ry 0 rz 19.31 deg; joints [136.509, -12.198, 21.35, -98.581, 47.198, 115.28, 25, -19.31]
  MoveL 498 to (-33.02, 86.8, 119.09) mm, rotated rx 142.24 ry 0 rz 19.31 deg; joints [136.477, -12.236, 21.392, -98.594, 47.166, 115.292, 25, -19.31]
  MoveL 499 to (-33.05, 87.15, 118.83) mm, rotated rx 142.08 ry 0 rz 19.26 deg; joints [136.43, -12.301, 21.463, -98.612, 47.121, 115.47, 25, -19.259]
  MoveL 500 to (-33.06, 87.43, 118.62) mm, rotated rx 142.08 ry 0 rz 19.26 deg; joints [136.424, -12.315, 21.477, -98.614, 47.116, 115.472, 25, -19.259]
  MoveL 501 to (-32.96, 88.58, 117.78) mm, rotated rx 141.57 ry 0 rz 18.98 deg; joints [136.278, -12.516, 21.695, -98.673, 46.976, 116.028, 25, -18.98]
  MoveL 502 to (-32.9, 88.59, 117.79) mm, rotated rx 140.37 ry 0 rz 20.86 deg; joints [136.082, -12.994, 22.19, -98.748, 46.787, 117.3, 25, -20.863]
  MoveL 503 to (-33.33, 88.3, 117.9) mm, rotated rx 140.55 ry 0 rz 21.55 deg; joints [136.144, -12.953, 22.138, -98.72, 46.846, 117.091, 25, -21.554]
  MoveL 504 to (-33.48, 88.12, 117.99) mm, rotated rx 140.6 ry 0 rz 21.68 deg; joints [136.16, -12.931, 22.114, -98.713, 46.861, 117.03, 25, -21.676]
  MoveL 505 to (-35.76, 84.84, 119.71) mm, rotated rx 141.71 ry 0 rz 23.85 deg; joints [136.481, -12.5, 21.645, -98.582, 47.169, 115.807, 25, -23.846]
  Set speed (16.7 mm/s)
  MoveL 506 to (-40.78, 96.17, 135.41) mm, rotated rx 141.71 ry 0 rz 23.85 deg; joints [136.371, -12.679, 21.097, -97.944, 46.956, 114.846, 25, -23.846]
  Set speed (1000.0 mm/s)
  MoveL 507 to (-45.17, 95.45, 134.52) mm, rotated rx 141.64 ry 0 rz 24.02 deg; joints [136.221, -12.621, 21.066, -98.011, 46.813, 114.982, 25, -24.021]
  Set speed (5.0 mm/s)
  MoveL 508 to (-40.12, 84.12, 118.84) mm, rotated rx 141.64 ry 0 rz 24.02 deg; joints [136.332, -12.441, 21.612, -98.651, 47.027, 115.944, 25, -24.021]
  Set speed (16.7 mm/s)
  MoveL 509 to (-43.3, 87.22, 115.43) mm, rotated rx 139.58 ry 0 rz 25 deg; joints [135.733, -13.252, 22.506, -98.908, 46.455, 118.238, 25, -24.997]
  MoveL 510 to (-43.57, 87.55, 115.08) mm, rotated rx 139.58 ry 0 rz 25 deg; joints [135.718, -13.266, 22.522, -98.915, 46.441, 118.245, 25, -24.997]
  MoveL 511 to (-43.75, 87.84, 114.79) mm, rotated rx 139.41 ry 0 rz 25.02 deg; joints [135.668, -13.332, 22.596, -98.937, 46.394, 118.435, 25, -25.017]
  MoveL 512 to (-43.84, 88.04, 114.6) mm, rotated rx 139.41 ry 0 rz 25.02 deg; joints [135.661, -13.341, 22.606, -98.941, 46.387, 118.438, 25, -25.017]
  MoveL 513 to (-44.64, 90.03, 112.73) mm, rotated rx 138.33 ry 0 rz 24.95 deg; joints [135.345, -13.758, 23.077, -99.09, 46.087, 119.655, 25, -24.949]
  MoveL 514 to (-44.6, 90.01, 112.76) mm, rotated rx 137.53 ry 0 rz 25.54 deg; joints [135.186, -14.035, 23.382, -99.166, 45.937, 120.529, 25, -25.538]
  MoveL 515 to (-47.82, 90.06, 111.4) mm, rotated rx 136.76 ry 0 rz 27.16 deg; joints [134.956, -14.332, 23.725, -99.283, 45.721, 121.42, 25, -27.163]
  MoveL 516 to (-48.39, 90.12, 111.1) mm, rotated rx 136.76 ry 0 rz 27.16 deg; joints [134.934, -14.33, 23.728, -99.296, 45.699, 121.433, 25, -27.163]
  MoveL 517 to (-48.53, 90.16, 111.01) mm, rotated rx 136.71 ry 0 rz 27.22 deg; joints [134.919, -14.348, 23.75, -99.303, 45.686, 121.489, 25, -27.224]
  MoveL 518 to (-49.07, 90.37, 110.6) mm, rotated rx 136.71 ry 0 rz 27.22 deg; joints [134.895, -14.354, 23.761, -99.316, 45.663, 121.502, 25, -27.224]
  MoveL 519 to (-50.17, 91.04, 109.55) mm, rotated rx 136.12 ry 0 rz 27.6 deg; joints [134.722, -14.576, 24.021, -99.408, 45.5, 122.179, 25, -27.601]
  MoveL 520 to (-50.02, 90.97, 109.68) mm, rotated rx 136.01 ry 0 rz 27.7 deg; joints [134.706, -14.613, 24.061, -99.416, 45.486, 122.298, 25, -27.696]
  MoveL 521 to (-51.81, 91.46, 108.44) mm, rotated rx 135.32 ry 0 rz 28.45 deg; joints [134.502, -14.873, 24.368, -99.529, 45.295, 123.102, 25, -28.451]
  MoveL 522 to (-52.18, 91.59, 108.14) mm, rotated rx 135.32 ry 0 rz 28.45 deg; joints [134.485, -14.877, 24.377, -99.539, 45.279, 123.112, 25, -28.451]
  MoveL 523 to (-52.78, 92.16, 107.37) mm, rotated rx 135.32 ry 0 rz 28.45 deg; joints [134.452, -14.902, 24.409, -99.557, 45.248, 123.131, 25, -28.451]
  MoveL 524 to (-53.01, 92.57, 106.9) mm, rotated rx 135.07 ry 0 rz 28.45 deg; joints [134.376, -14.996, 24.522, -99.6, 45.178, 123.426, 25, -28.452]
  MoveL 525 to (-53.17, 93.2, 106.27) mm, rotated rx 135.07 ry 0 rz 28.45 deg; joints [134.359, -15.028, 24.559, -99.61, 45.162, 123.436, 25, -28.452]
  MoveL 526 to (-53.1, 96.96, 102.89) mm, rotated rx 133.3 ry 0 rz 27.5 deg; joints [133.827, -15.683, 25.354, -99.928, 44.669, 125.53, 25, -27.502]
  MoveL 527 to (-52.96, 97.63, 102.33) mm, rotated rx 131.79 ry 0 rz 27.96 deg; joints [133.483, -16.181, 25.954, -100.148, 44.352, 127.265, 25, -27.959]
  MoveL 528 to (-54.46, 97.31, 101.85) mm, rotated rx 131.54 ry 0 rz 28.72 deg; joints [133.407, -16.271, 26.067, -100.197, 44.284, 127.566, 25, -28.722]
  MoveL 529 to (-55.01, 97.23, 101.62) mm, rotated rx 131.54 ry 0 rz 28.72 deg; joints [133.387, -16.262, 26.065, -100.211, 44.265, 127.58, 25, -28.722]
  MoveL 530 to (-56.07, 97.47, 100.81) mm, rotated rx 131.54 ry 0 rz 28.72 deg; joints [133.34, -16.265, 26.082, -100.242, 44.222, 127.612, 25, -28.722]
  MoveL 531 to (-56.25, 97.58, 100.61) mm, rotated rx 131.44 ry 0 rz 28.78 deg; joints [133.309, -16.302, 26.129, -100.263, 44.194, 127.737, 25, -28.776]
  MoveL 532 to (-56.8, 98.31, 99.58) mm, rotated rx 131.44 ry 0 rz 28.78 deg; joints [133.272, -16.337, 26.176, -100.288, 44.16, 127.763, 25, -28.776]
  MoveL 533 to (-57.06, 99.51, 98.22) mm, rotated rx 130.76 ry 0 rz 28.6 deg; joints [133.067, -16.577, 26.484, -100.429, 43.974, 128.586, 25, -28.604]
  MoveL 534 to (-57.33, 99.74, 97.84) mm, rotated rx 130.61 ry 0 rz 28.62 deg; joints [133.016, -16.631, 26.554, -100.464, 43.927, 128.774, 25, -28.621]
  MoveL 535 to (-57.59, 100.47, 96.93) mm, rotated rx 130.27 ry 0 rz 28.66 deg; joints [132.911, -16.767, 26.726, -100.539, 43.831, 129.195, 25, -28.66]
  MoveL 536 to (-57.51, 102.68, 94.63) mm, rotated rx 129.14 ry 0 rz 28.11 deg; joints [132.569, -17.158, 27.239, -100.789, 43.523, 130.582, 25, -28.113]
  Set speed (16.7 mm/s)
  MoveL 537 to (-64.82, 116.37, 107.26) mm, rotated rx 129.14 ry 0 rz 28.11 deg; joints [132.33, -17.476, 26.839, -100.126, 43.161, 129.615, 25, -28.113]
  Set speed (1000.0 mm/s)
  MoveL 538 to (-61.57, 118.93, 106.35) mm, rotated rx 129.16 ry 0 rz 27.96 deg; joints [132.397, -17.636, 26.976, -100.079, 43.223, 129.552, 25, -27.955]
  Set speed (5.0 mm/s)
  MoveL 539 to (-54.3, 105.24, 93.72) mm, rotated rx 129.16 ry 0 rz 27.96 deg; joints [132.637, -17.317, 27.377, -100.742, 43.585, 130.52, 25, -27.955]
  Set speed (16.7 mm/s)
  MoveL 540 to (-52.25, 105.41, 94.68) mm, rotated rx 129.62 ry 0 rz 27.04 deg; joints [132.778, -17.156, 27.164, -100.637, 43.713, 129.944, 25, -27.037]
  MoveL 541 to (-52.32, 105.39, 94.67) mm, rotated rx 129.76 ry 0 rz 26.54 deg; joints [132.784, -17.08, 27.085, -100.633, 43.717, 129.799, 25, -26.535]
  MoveL 542 to (-50.68, 106.06, 94.82) mm, rotated rx 129.84 ry 0 rz 25.68 deg; joints [132.806, -17.054, 27.052, -100.616, 43.737, 129.708, 25, -25.675]
  MoveL 543 to (-50.29, 106.19, 94.87) mm, rotated rx 129.85 ry 0 rz 25.57 deg; joints [132.816, -17.055, 27.049, -100.609, 43.746, 129.685, 25, -25.569]
  MoveL 544 to (-48.62, 106.73, 95.14) mm, rotated rx 129.99 ry 0 rz 24.59 deg; joints [132.853, -16.996, 26.977, -100.582, 43.779, 129.513, 25, -24.592]
  MoveL 545 to (-48.14, 106.92, 95.18) mm, rotated rx 130.01 ry 0 rz 24.34 deg; joints [132.857, -16.991, 26.97, -100.579, 43.784, 129.493, 25, -24.34]
  MoveL 546 to (-44.06, 108.2, 95.7) mm, rotated rx 130.26 ry 0 rz 22.36 deg; joints [132.939, -16.909, 26.86, -100.52, 43.858, 129.181, 25, -22.357]
  MoveL 547 to (-42.82, 108.32, 96.12) mm, rotated rx 130.26 ry 0 rz 22.36 deg; joints [132.983, -16.935, 26.872, -100.49, 43.897, 129.15, 25, -22.357]
  MoveL 548 to (-42.06, 108.1, 96.71) mm, rotated rx 130.26 ry 0 rz 22.36 deg; joints [133.017, -16.935, 26.86, -100.466, 43.928, 129.125, 25, -22.357]
  MoveL 549 to (-41.68, 107.78, 97.23) mm, rotated rx 130.26 ry 0 rz 22.36 deg; joints [133.04, -16.924, 26.841, -100.45, 43.949, 129.108, 25, -22.357]
  MoveL 550 to (-41.44, 107.16, 98.02) mm, rotated rx 130.26 ry 0 rz 22.36 deg; joints [133.065, -16.893, 26.803, -100.433, 43.972, 129.09, 25, -22.357]
  MoveL 551 to (-41.61, 106.43, 98.74) mm, rotated rx 130.26 ry 0 rz 22.36 deg; joints [133.077, -16.851, 26.756, -100.424, 43.982, 129.081, 25, -22.357]
  MoveL 552 to (-41.91, 105.85, 99.24) mm, rotated rx 130.51 ry 0 rz 22.61 deg; joints [133.153, -16.762, 26.642, -100.371, 44.052, 128.773, 25, -22.607]
  MoveL 553 to (-42.02, 105.65, 99.4) mm, rotated rx 130.51 ry 0 rz 22.61 deg; joints [133.154, -16.75, 26.629, -100.37, 44.052, 128.772, 25, -22.607]
  MoveL 554 to (-42.66, 104.64, 100.19) mm, rotated rx 130.92 ry 0 rz 23.11 deg; joints [133.276, -16.608, 26.447, -100.287, 44.163, 128.283, 25, -23.106]
  MoveL 555 to (-42.71, 104.67, 100.13) mm, rotated rx 132.48 ry 0 rz 22.07 deg; joints [133.593, -16.098, 25.837, -100.075, 44.454, 126.501, 25, -22.074]
  MoveL 556 to (-42.56, 104.75, 100.12) mm, rotated rx 132.47 ry 0 rz 22.01 deg; joints [133.593, -16.101, 25.841, -100.075, 44.454, 126.506, 25, -22.011]
  MoveL 557 to (-40.52, 105.67, 99.99) mm, rotated rx 132.41 ry 0 rz 20.88 deg; joints [133.573, -16.125, 25.871, -100.089, 44.435, 126.587, 25, -20.877]
  Set speed (16.7 mm/s)
  MoveL 558 to (-45.78, 119.47, 113.47) mm, rotated rx 132.41 ry 0 rz 20.88 deg; joints [133.369, -16.409, 25.431, -99.426, 44.114, 125.615, 25, -20.877]
  Set speed (1000.0 mm/s)
  MoveL 559 to (-43.02, 122.52, 111.29) mm, rotated rx 131.42 ry 0 rz 19.58 deg; joints [133.078, -16.798, 25.908, -99.611, 43.846, 126.797, 25, -19.582]
  Set speed (5.0 mm/s)
  MoveL 560 to (-38, 108.39, 98.06) mm, rotated rx 131.42 ry 0 rz 19.58 deg; joints [133.293, -16.504, 26.337, -100.274, 44.179, 127.768, 25, -19.582]
  Set speed (16.7 mm/s)
  MoveL 561 to (-35.84, 108.8, 98.41) mm, rotated rx 131.59 ry 0 rz 18.5 deg; joints [133.346, -16.441, 26.257, -100.238, 44.228, 127.555, 25, -18.498]
  MoveL 562 to (-35.69, 108.96, 98.29) mm, rotated rx 131.11 ry 0 rz 17.08 deg; joints [133.162, -16.488, 26.363, -100.363, 44.059, 128.165, 25, -17.076]
  MoveL 563 to (-35.48, 109.37, 97.91) mm, rotated rx 130.92 ry 0 rz 16.92 deg; joints [133.104, -16.556, 26.45, -100.403, 44.007, 128.397, 25, -16.918]
  MoveL 564 to (-34.6, 111.34, 95.98) mm, rotated rx 129.93 ry 0 rz 16.19 deg; joints [132.805, -16.899, 26.895, -100.615, 43.736, 129.608, 25, -16.193]
  MoveL 565 to (-36.6, 110.9, 95.75) mm, rotated rx 128.56 ry 0 rz 18.95 deg; joints [132.559, -17.407, 27.495, -100.801, 43.515, 131.176, 25, -18.948]
  MoveL 566 to (-38.39, 109.26, 96.92) mm, rotated rx 129.14 ry 0 rz 20.05 deg; joints [132.736, -17.207, 27.23, -100.669, 43.674, 130.456, 25, -20.054]
  MoveL 567 to (-39.39, 108.62, 97.25) mm, rotated rx 129.14 ry 0 rz 20.05 deg; joints [132.717, -17.155, 27.184, -100.681, 43.657, 130.469, 25, -20.054]
  MoveL 568 to (-40.02, 108.41, 97.23) mm, rotated rx 129.14 ry 0 rz 20.05 deg; joints [132.699, -17.132, 27.167, -100.694, 43.641, 130.482, 25, -20.054]
  MoveL 569 to (-40.83, 108.3, 97.01) mm, rotated rx 129.14 ry 0 rz 20.05 deg; joints [132.673, -17.112, 27.156, -100.713, 43.617, 130.502, 25, -20.054]
  MoveL 570 to (-41.87, 108.5, 96.34) mm, rotated rx 129.14 ry 0 rz 20.05 deg; joints [132.628, -17.104, 27.164, -100.745, 43.577, 130.536, 25, -20.054]
  MoveL 571 to (-42.38, 108.74, 95.85) mm, rotated rx 128.9 ry 0 rz 20.25 deg; joints [132.554, -17.188, 27.275, -100.8, 43.51, 130.838, 25, -20.248]
  MoveL 572 to (-42.97, 109.28, 94.96) mm, rotated rx 128.9 ry 0 rz 20.25 deg; joints [132.517, -17.207, 27.307, -100.828, 43.477, 130.867, 25, -20.248]
  MoveL 573 to (-43.02, 110.11, 93.98) mm, rotated rx 128.9 ry 0 rz 20.25 deg; joints [132.492, -17.25, 27.36, -100.847, 43.455, 130.887, 25, -20.248]
  MoveL 574 to (-42.61, 110.81, 93.34) mm, rotated rx 128.9 ry 0 rz 20.25 deg; joints [132.488, -17.296, 27.407, -100.851, 43.451, 130.892, 25, -20.248]
  MoveL 575 to (-39.45, 114.19, 90.61) mm, rotated rx 127.6 ry 0 rz 18.29 deg; joints [132.092, -17.739, 28.005, -101.16, 43.098, 132.52, 25, -18.294]
  MoveL 576 to (-38.76, 114.71, 90.25) mm, rotated rx 127.6 ry 0 rz 18.29 deg; joints [132.102, -17.78, 28.043, -101.154, 43.106, 132.514, 25, -18.294]
  MoveL 577 to (-38.14, 115.07, 90.06) mm, rotated rx 127.51 ry 0 rz 17.96 deg; joints [132.075, -17.81, 28.084, -101.176, 43.082, 132.626, 25, -17.96]
  MoveL 578 to (-32.45, 117.85, 88.68) mm, rotated rx 126.88 ry 0 rz 15.08 deg; joints [131.884, -18.028, 28.381, -101.333, 42.914, 133.427, 25, -15.082]
  MoveL 579 to (-31.78, 118.21, 88.45) mm, rotated rx 126.78 ry 0 rz 14.81 deg; joints [131.858, -18.067, 28.431, -101.354, 42.891, 133.547, 25, -14.812]
  MoveL 580 to (-27.47, 119.84, 87.7) mm, rotated rx 126.43 ry 0 rz 12.67 deg; joints [131.75, -18.184, 28.594, -101.444, 42.796, 133.995, 25, -12.674]
  Set speed (16.7 mm/s)
  MoveL 581 to (-31, 135.54, 99.57) mm, rotated rx 126.43 ry 0 rz 12.67 deg; joints [131.481, -18.531, 28.225, -100.784, 42.398, 133.034, 25, -12.674]
  Set speed (1000.0 mm/s)
  MoveL 582 to (-27.64, 135.23, 100.97) mm, rotated rx 126.99 ry 0 rz 11.24 deg; joints [131.652, -18.329, 27.953, -100.645, 42.551, 132.327, 25, -11.239]
  Set speed (5.0 mm/s)
  MoveL 583 to (-24.52, 119.56, 88.93) mm, rotated rx 126.99 ry 0 rz 11.24 deg; joints [131.915, -17.988, 28.328, -101.306, 42.942, 133.29, 25, -11.239]
  Set speed (16.7 mm/s)
  MoveL 584 to (-23.46, 119.99, 88.66) mm, rotated rx 126.85 ry 0 rz 10.71 deg; joints [131.875, -18.032, 28.389, -101.339, 42.906, 133.458, 25, -10.712]
  MoveL 585 to (-22.96, 120.18, 88.53) mm, rotated rx 126.7 ry 0 rz 10.2 deg; joints [131.82, -18.057, 28.436, -101.384, 42.858, 133.66, 25, -10.203]
  MoveL 586 to (-16.96, 123.4, 85.38) mm, rotated rx 125.24 ry 0 rz 7.23 deg; joints [131.377, -18.535, 29.108, -101.766, 42.47, 135.525, 25, -7.234]
  MoveL 587 to (-16.95, 123.4, 85.38) mm, rotated rx 124.49 ry 0 rz 6.67 deg; joints [131.167, -18.682, 29.35, -101.953, 42.287, 136.48, 25, -6.673]
  MoveL 588 to (-16.96, 123.93, 84.62) mm, rotated rx 124.14 ry 0 rz 6.65 deg; joints [131.06, -18.794, 29.512, -102.052, 42.195, 136.937, 25, -6.648]
  MoveL 589 to (-16.68, 124.61, 83.67) mm, rotated rx 124.14 ry 0 rz 6.65 deg; joints [131.041, -18.836, 29.565, -102.071, 42.178, 136.958, 25, -6.648]
  MoveL 590 to (-15.89, 125.18, 82.97) mm, rotated rx 124.14 ry 0 rz 6.65 deg; joints [131.041, -18.889, 29.62, -102.073, 42.179, 136.961, 25, -6.648]
  MoveL 591 to (-15.74, 125.26, 82.89) mm, rotated rx 124.1 ry 0 rz 6.58 deg; joints [131.03, -18.9, 29.636, -102.083, 42.17, 137.007, 25, -6.576]
  MoveL 592 to (-14.94, 125.53, 82.63) mm, rotated rx 124.1 ry 0 rz 6.58 deg; joints [131.043, -18.939, 29.671, -102.073, 42.181, 136.997, 25, -6.576]
  MoveL 593 to (-11.91, 126.15, 82.16) mm, rotated rx 123.81 ry 0 rz 4.9 deg; joints [130.945, -19.002, 29.78, -102.164, 42.096, 137.384, 25, -4.897]
  MoveL 594 to (-8.8, 127.24, 80.87) mm, rotated rx 123.23 ry 0 rz 3.46 deg; joints [130.768, -19.184, 30.049, -102.332, 41.946, 138.146, 25, -3.465]
  MoveL 595 to (-8.25, 127.38, 80.71) mm, rotated rx 123.23 ry 0 rz 3.46 deg; joints [130.778, -19.209, 30.071, -102.325, 41.954, 138.139, 25, -3.465]
  MoveL 596 to (-8.04, 127.41, 80.67) mm, rotated rx 123.22 ry 0 rz 3.37 deg; joints [130.772, -19.215, 30.079, -102.33, 41.949, 138.162, 25, -3.369]
  MoveL 597 to (-7.82, 127.45, 80.64) mm, rotated rx 123.22 ry 0 rz 3.37 deg; joints [130.777, -19.224, 30.087, -102.326, 41.953, 138.158, 25, -3.369]
  MoveL 598 to (-6.62, 127.59, 80.51) mm, rotated rx 123.16 ry 0 rz 2.83 deg; joints [130.759, -19.242, 30.114, -102.343, 41.938, 138.234, 25, -2.827]
  MoveL 599 to (-6.62, 127.59, 80.53) mm, rotated rx 122.88 ry 0 rz 2.16 deg; joints [130.657, -19.253, 30.173, -102.438, 41.851, 138.611, 25, -2.159]
  MoveL 600 to (-4.42, 128.9, 78.57) mm, rotated rx 122.01 ry 0 rz 1.16 deg; joints [130.392, -19.522, 30.58, -102.703, 41.626, 139.773, 25, -1.163]
  MoveL 601 to (-3.96, 129.11, 78.25) mm, rotated rx 122.01 ry 0 rz 1.16 deg; joints [130.394, -19.549, 30.606, -102.703, 41.629, 139.773, 25, -1.163]
  MoveL 602 to (-3.78, 129.17, 78.15) mm, rotated rx 121.96 ry 0 rz 1.08 deg; joints [130.38, -19.562, 30.627, -102.717, 41.617, 139.833, 25, -1.078]
  MoveL 603 to (-3.52, 129.26, 78.02) mm, rotated rx 121.96 ry 0 rz 1.08 deg; joints [130.383, -19.576, 30.64, -102.715, 41.62, 139.831, 25, -1.078]
  MoveL 604 to (-1.85, 129.7, 77.34) mm, rotated rx 121.66 ry 0 rz 0.34 deg; joints [130.292, -19.667, 30.78, -102.808, 41.543, 140.234, 25, -0.341]
  MoveL 605 to (-1.88, 129.69, 77.35) mm, rotated rx 121.39 ry 0 rz 0 deg; joints [130.207, -19.702, 30.858, -102.893, 41.472, 140.599, 25, 0]
  MoveL 606 to (0.05, 130.9, 75.32) mm, rotated rx 120.52 ry 0 rz -0.87 deg; joints [129.941, -19.96, 31.265, -103.175, 41.251, 141.777, 25, 0.868]
  MoveL 607 to (2.04, 131.33, 74.53) mm, rotated rx 119.6 ry 0 rz -1.98 deg; joints [129.689, -20.171, 31.619, -103.451, 41.043, 142.991, 25, 1.979]
  MoveL 608 to (2.19, 133.01, 71.49) mm, rotated rx 118.28 ry 0 rz -2.02 deg; joints [129.292, -20.548, 32.236, -103.905, 40.722, 144.809, 25, 2.019]
  MoveL 609 to (2.5, 133.53, 70.5) mm, rotated rx 118.28 ry 0 rz -2.02 deg; joints [129.273, -20.584, 32.286, -103.93, 40.707, 144.836, 25, 2.019]
  MoveL 610 to (3.29, 133.91, 69.74) mm, rotated rx 118.28 ry 0 rz -2.02 deg; joints [129.271, -20.633, 32.34, -103.936, 40.706, 144.844, 25, 2.019]
  MoveL 611 to (3.86, 134.08, 69.39) mm, rotated rx 118.13 ry 0 rz -2.26 deg; joints [129.226, -20.675, 32.41, -103.989, 40.67, 145.052, 25, 2.262]
  MoveL 612 to (4.1, 134.14, 69.26) mm, rotated rx 118.13 ry 0 rz -2.26 deg; joints [129.228, -20.688, 32.422, -103.988, 40.673, 145.05, 25, 2.262]
  MoveL 613 to (10, 135.24, 66.47) mm, rotated rx 116.95 ry 0 rz -4.73 deg; joints [128.876, -21.013, 32.974, -104.417, 40.395, 146.701, 25, 4.727]
  MoveL 614 to (10.53, 135.3, 66.25) mm, rotated rx 116.88 ry 0 rz -4.9 deg; joints [128.857, -21.038, 33.013, -104.442, 40.38, 146.798, 25, 4.896]
  MoveL 615 to (10.74, 135.32, 66.18) mm, rotated rx 116.88 ry 0 rz -4.9 deg; joints [128.86, -21.048, 33.021, -104.439, 40.382, 146.796, 25, 4.896]
  MoveL 616 to (14.37, 135.54, 65.03) mm, rotated rx 116.29 ry 0 rz -6.65 deg; joints [128.677, -21.178, 33.272, -104.667, 40.239, 147.639, 25, 6.654]
  MoveL 617 to (17.64, 136.09, 63.05) mm, rotated rx 115.46 ry 0 rz -7.98 deg; joints [128.433, -21.396, 33.659, -104.985, 40.052, 148.814, 25, 7.978]
  MoveL 618 to (17.92, 136.12, 62.91) mm, rotated rx 115.46 ry 0 rz -7.98 deg; joints [128.436, -21.41, 33.673, -104.983, 40.054, 148.813, 25, 7.978]
  MoveL 619 to (18.45, 136.16, 62.66) mm, rotated rx 115.36 ry 0 rz -8.19 deg; joints [128.406, -21.436, 33.719, -105.022, 40.032, 148.956, 25, 8.193]
  MoveL 620 to (18.4, 136.15, 62.7) mm, rotated rx 115.14 ry 0 rz -8.49 deg; joints [128.339, -21.448, 33.776, -105.107, 39.98, 149.263, 25, 8.495]
  MoveL 621 to (23.58, 137.65, 57.46) mm, rotated rx 112.98 ry 0 rz -10.5 deg; joints [127.709, -21.988, 34.786, -105.988, 39.513, 152.39, 25, 10.501]
  MoveL 622 to (23.57, 137.63, 57.51) mm, rotated rx 112.16 ry 0 rz -10.71 deg; joints [127.509, -22.121, 35.073, -106.278, 39.369, 153.536, 25, 10.711]
  MoveL 623 to (23.29, 138.27, 56.09) mm, rotated rx 111.57 ry 0 rz -10.55 deg; joints [127.341, -22.257, 35.345, -106.531, 39.251, 154.397, 25, 10.551]
  MoveL 624 to (23.25, 138.42, 55.74) mm, rotated rx 111.57 ry 0 rz -10.55 deg; joints [127.331, -22.262, 35.357, -106.546, 39.243, 154.414, 25, 10.551]
  MoveL 625 to (23.25, 138.49, 55.57) mm, rotated rx 111.5 ry 0 rz -10.54 deg; joints [127.312, -22.278, 35.389, -106.576, 39.23, 154.515, 25, 10.545]
  MoveL 626 to (23.25, 138.58, 55.33) mm, rotated rx 111.5 ry 0 rz -10.54 deg; joints [127.305, -22.282, 35.398, -106.585, 39.225, 154.525, 25, 10.545]
  MoveL 627 to (23.37, 139.11, 53.93) mm, rotated rx 110.94 ry 0 rz -10.55 deg; joints [127.143, -22.411, 35.663, -106.837, 39.113, 155.37, 25, 10.551]
  MoveL 628 to (23.32, 139.35, 53.34) mm, rotated rx 110.71 ry 0 rz -10.52 deg; joints [127.078, -22.463, 35.77, -106.94, 39.068, 155.711, 25, 10.516]
  MoveL 629 to (23.65, 140.64, 49.68) mm, rotated rx 109.23 ry 0 rz -10.55 deg; joints [126.661, -22.785, 36.458, -107.619, 38.79, 157.937, 25, 10.551]
  MoveL 630 to (24.07, 140.97, 48.53) mm, rotated rx 109.23 ry 0 rz -10.55 deg; joints [126.642, -22.82, 36.513, -107.655, 38.779, 157.978, 25, 10.551]
  MoveL 631 to (24.75, 141.09, 47.85) mm, rotated rx 109.23 ry 0 rz -10.55 deg; joints [126.641, -22.858, 36.558, -107.663, 38.78, 157.988, 25, 10.551]
  MoveL 632 to (25.64, 141.06, 47.45) mm, rotated rx 109.23 ry 0 rz -10.55 deg; joints [126.653, -22.902, 36.599, -107.653, 38.79, 157.978, 25, 10.551]
  MoveL 633 to (26.99, 140.8, 47.48) mm, rotated rx 109.23 ry 0 rz -10.55 deg; joints [126.687, -22.957, 36.636, -107.61, 38.816, 157.935, 25, 10.551]
  MoveL 634 to (27.66, 140.6, 47.69) mm, rotated rx 109.31 ry 0 rz -10.83 deg; joints [126.71, -22.94, 36.598, -107.571, 38.831, 157.808, 25, 10.832]
